METHOD Initialization : BOOL
VAR_INPUT
	_Testmode	: BOOL;
END_VAR

VAR
	bConfig: BOOL;
END_VAR
(*
_tmrT0(IN:=TRUE,PT:=T#0.2S);
LoadCell.i_bCmd_Tara:= NOT _tmrT0.Q  ;
Initialization	:= AssRoller.Initialization() AND _tmrT0.Q ;
SamplingWeight	:=0;
Cyl_NGPurge.qExtendCoil	:= FALSE;
Roller_Purge.qRun:= FALSE;
Motor_shock.qRun	:= FALSE;
Motor_shock.qSign	:= FALSE;
Cyl_ShockStop.qExtendCoil:= FALSE;
*)

_bInitialScan:=TRUE;

CASE nInitiStep OF
	0:		
		LoadCell.GetTara();
		_tmrT0(IN:=FALSE);
		strText:='ORG : Initial ';
		Cyl_NGPurge.qExtendCoil		:= FALSE;
		Roller_Purge.qRun			:= FALSE;
		Motor_shock.qRun			:= FALSE;
		Motor_shock.qSign			:= FALSE;
		Cyl_ShockStop.qExtendCoil	:= FALSE;		
		nInitiStep						:= 5;
	5:
		bConfig			:=TRUE;
		IF Sen_TFLoadIn THEN
			bConfig			:=FALSE;
			EventLogger.eEventType		:= 3;
			EventLogger.strEventText	:= 'TF Sensor Error ';	
			EventLogger();					
		END_IF		
			
		IF bConfig THEN
			nInitiStep	:= 10;
			strText:='ORG : Runing ';
			ELSE
			strText:='ORG : Failed ';
			nInitiStep	:= 50;
		END_IF	
	10:
		IF AssRoller.Initialization() THEN
			strText		:='ORG : Done ';
			nInitiStep	:= 20;
		END_IF;		
	20:
		Initialization	:= TRUE;
	
END_CASE;
END_METHOD

{warning 'add property implementation'}
PROPERTY NoEntry : BOOL
GET
END_GET
END_PROPERTY

{warning 'add method implementation '}
METHOD Pause : BOOL
END_METHOD

METHOD Process : BOOL
VAR_INPUT
	bHlatMode	: BOOL;
END_VAR

VAR
	bStoppedComv: BOOL;
END_VAR
_bProcessScan:= TRUE;
//判斷 

CASE nStep OF
	0:
		tmrLoadcell(IN:= FALSE);
		_tmrT0(IN:=FALSE);
		AssRoller.Roller();
		strText:= 'Waiting';
		IF Sen_TFLoadIn THEN
			nStep := 5;
		END_IF
	5:
		strText:= 'Loadind and Stop';
		AssRoller.Roller();
		IF NOT Sen_TFLoadIn THEN
			SamplingWeight	:= 0;
			nStep := 10;
		END_IF	
	10:		
		strText:= 'Weight Check!';
		tmrLoadcell(IN:= TRUE,PT:=T#1S);
		UpperWeight	:= RunParameter.PackagingWeight + RunParameter.PackagingWeightUpLimit ;
		LowerWeight := RunParameter.PackagingWeight - RunParameter.PackagingWeightLowLimit ;
		IF tmrLoadcell.Q THEN
			tmrLoadcell(IN:= FALSE,PT:=T#1S);
			SamplingWeight	:= 	LoadCell.o_rWeight;
			IF SamplingWeight >= LowerWeight AND
				SamplingWeight <= UpperWeight THEN
				strText:= 'Weight Pass!';
				bBoxPass:= TRUE;
				ELSE
				EventLogger.eEventType		:= 2;
				EventLogger.strEventText	:= 'Box Over Weight ';	
				EventLogger.strEventText	:=	CONCAT(EventLogger.strEventText,LEFT(REAL_TO_STRING(SamplingWeight),3));
				EventLogger();
				strText:= 'Box NG';
				bBoxPass:= FALSE;
			END_IF
			nStep := 15;
		END_IF
	
	15:
		
		IF nNGstep = 0 THEN
			nNGstep	:= 5;
			IF RunParameter.PackagingCheck THEN
				bStoppedComv	:= TRUE;
			END_IF
			AssRoller.Belt();
			IF Sen_NGLoadOut THEN
				nStep := 0;
			END_IF;
		END_IF
		
		
		
		
END_CASE;

CASE nNGstep OF
	0:
		strNGText	:= 'Wait BOX';
		tmrNG(IN:=FALSE,PT:=T#2S);
		Roller_Purge.qRun:= TRUE;
		IF Sen_NGLoadOut THEN
			strNGText	:= 'Active Loading';
			nNGstep := 20;
			CASE nStep OF
				0..10:
				strNGText	:= 'Up Loading';
				nNGstep := 50;
			END_CASE
		END_IF
	5:
		strNGText	:= 'TF Loading';
		AssRoller.Belt();
	
		IF Sen_NGLoadOut THEN
			nStep := 0;
			nNGstep	:= 6;
		END_IF
	6:
			IF bBoxPass THEN
				strNGText	:= 'TF LoadIn Stop';
				Roller_Purge.qRun:= FALSE;
				nStep := 0;
				IF nShackStep = 1 THEN
					strNGText	:= 'Go Shack';
					Roller_Purge.qRun:= TRUE;
					nNGstep	:= 10;
				END_IF;
				ELSE
				EventLogger.eEventType		:= 2;
				EventLogger.strEventText	:= 'NG Perge!';		
				EventLogger();		
				strNGText	:= 'TF NG Perge';
				nNGstep	:= 30;
				Roller_Purge.qRun:= FALSE;
			END_IF		

		
	10:
		IF Sen_ShockPos THEN
			strNGText	:= 'Shack ORG';
			nNGstep	:= 0;
		END_IF
	
	
	30://重量Error
		Cyl_NGPurge.qExtendCoil	:= TRUE;
		tmrNG(IN:=TRUE,PT:=T#2S);
		IF tmrNG.Q THEN
			tmrNG(IN:=FALSE);
			nStep := 0;
			Cyl_NGPurge.qExtendCoil	:= FALSE;
			nNGstep := 0;
		END_IF		
		
		
		
	50://手動投入	
		strNGText	:= '50 Man. ';
		IF Sen_ShockPos THEN
			nNGstep	:= 0;
		END_IF	
END_CASE;	
CASE nShackStep OF
	0:
		tmrshock(IN:=FALSE);
		nShackStep	:= 1;
	1:
		strShackText:='Wait Box';
		Cyl_ShockStop.qExtendCoil:= TRUE;
		tmrshock(IN:=Sen_ShockPos , PT:= RunParameter.shock_DelayTime);	
		Motor_shock.qRun	:= TRUE;
		Motor_shock.qSign	:= TRUE;
		IF tmrshock.q THEN
			strShackText:='Loading Box';
			tmrshock(IN:=FALSE);
			nShackStep	:= 5;
		END_IF
	5:
		strShackText:='Shack Box';
		Motor_shock.qSign	:= FALSE;
		tmrshock(IN:= TRUE, PT:= RunParameter.shock_HighTime);
		IF tmrshock.Q THEN
			tmrshock(IN:= FALSE);
			Motor_shock.qSign	:= TRUE;
			Cyl_ShockStop.qExtendCoil:= FALSE;
			nShackStep	:= 10;
		END_IF
	10:
		strShackText:='Load Out Box';
		tmrshock(IN:= NOT Sen_ShockPos , PT:= T#3S);				

		IF tmrshock.Q THEN
			Cyl_ShockStop.qExtendCoil:= TRUE;
			tmrshock(IN:= FALSE);
			nShackStep	:= 0;
		END_IF
		
		
END_CASE;
END_METHOD

PROPERTY Status : STRING(50)
GET
Status:= strText;
END_GET
END_PROPERTY

END_FUNCTION_BLOCK

// ---- 02_Unit/01_Customization/Ass_DualServo.TcPOU
FUNCTION_BLOCK Ass_DualServo IMPLEMENTS ITF_AutoStructCommand
VAR_INPUT
END_VAR
VAR_OUTPUT
END_VAR
VAR
	strText,strLeftText,strRightText	:STRING;
	tmrAuto	:TON:= (PT := TIME#1S0MS);
	bConfig	,_bError	:BOOL;
	_tmrT0		: TON;
	nInitiStep,nStopStep: INT;
	fb1_Stop,fb2_Stop,fbFly_Stop		:MC_Stop;
	fb1_Reset,fb2_Reset,fbFly_Reset		:MC_Reset;
	fbMC_MoveVelocityDaul: MC_MoveVelocity := (Velocity := 500);
	fbMC_GearIn: MC_GearIn;
	fbMC_GearOut: MC_GearOut;
	bDual1First,bDual2First,bDual1Done,bDual2Done	:BOOL;	
	MC_SetPositionLeft,MC_SetPositionRight,MC_SetPositionCon:MC_SetPosition;
	PreDual1Pos,PreDual2Pos	:  LREAL;
	L_Home,R_Home:MC_Home := (HomingMode := MC_HOMINGMODE.MC_ForceCalibration);
	MC_GroupReset: MC_GroupReset;
	LatchDual1Pos,LatchDual2Pos: LREAL;
	fbMC_MoveModule1,fbMC_MoveModule2	:MC_MoveModulo := (Velocity := 500);
	ConvQty	:INT;
	_bInitialScan	:BOOL;
	
	//Group
	fbMC_UngroupAllAxes	: MC_UngroupAllAxes;
	fbMC_GroupDisable	: MC_GroupDisable;
	fbAddAxis			: ARRAY[1..2] OF MC_AddAxisToGroup;
	fbMC_GroupEnable	: MC_GroupEnable;	
	fbMC_MoveAbsoluteCA_Left,fbMC_MoveAbsoluteCA_Right: MC_MoveAbsoluteCA := (Options := (GapControlMode := MC_GAP_CONTROL_MODE.mcGapControlModeFast));
	fbMC_GearInPosCA_Left,fbMC_GearInPosCA_Right		:MC_GearInPosCA;	
	nStep,nLeftStep,nRightStep,i	:INT;
	LeftLoadinQty,RifgtLoadinQty: UINT;
	bHMITriggerBtn: BOOL;
	fbMC_StopFly		:MC_Stop;
	MC_TouchProbeDual1,MC_TouchProbeDual2,MC_TouchProbeFly: MC_TouchProbe;
	TouchTriggerDual1,TouchTriggerDual2,TouchTriggerFly	:TRIGGER_REF;
	MC_AbortTrigger1,MC_AbortTrigger2					: MC_AbortTrigger;
	tmrT0,tmrT1	:TON := (ET := TIME#2S0MS);
	tmrFlyinDef	:TON;
	bPosfix	:BOOL;
	_bProcessScan: BOOL;
	_Dual1CalibrationPos , _Dual2CalibrationPos,_FlyInCalibrationPos	:LREAL;
	//
	fbSensorTrigger	:R_TRIG;
	dwSenesorTriggerTimes	:DWORD;
	
	wSlot: INT;
	bPause: BOOL;
	fRampTime: REAL;

END_VAR

Instance();
fbSensorTrigger(CLK:=Axis_FlyIn.DI.19);
IF fbSensorTrigger.Q THEN
	dwSenesorTriggerTimes	:= dwSenesorTriggerTimes+1;
END_IF



//Modhed
IF NOT _bProcessScan AND NOT _bInitialScan THEN
	MC_TouchProbeDual1.Execute	:= FALSE;
	MC_TouchProbeDual2.Execute	:= FALSE;
	strText:=strLeftText:=strRightText:='';
END_IF


IF NOT _bInitialScan THEN
	nInitiStep	:= 0;
END_IF

_bInitialScan:=FALSE;



IF NOT _bProcessScan THEN
	nStep	:= 0;
	nLeftStep	:=0;
	nRightStep	:=0;
END_IF


_bProcessScan:=FALSE;

METHOD _Clearfb : BOOL
VAR_INPUT
END_VAR
fbAddAxis[1](AxesGroup:=DualGroupRef, Axis := Axis_DualServo1, Execute := FALSE);
fbAddAxis[2](AxesGroup:=DualGroupRef, Axis := Axis_DualServo2, Execute := FALSE);
fbMC_MoveVelocityDaul(Axis:= Axis_DualServo1,Execute:= FALSE);
fbMC_GroupEnable(AxesGroup:= DualGroupRef, Execute:= FALSE);
fbMC_GroupDisable(AxesGroup:= DualGroupRef, Execute:= FALSE);	
fbMC_UngroupAllAxes(AxesGroup:= DualGroupRef,Execute:= FALSE);
fbMC_MoveAbsoluteCA_Left(Axis:= Axis_DualServo1,Execute:=FALSE);
fbMC_MoveAbsoluteCA_Right(Axis:= Axis_DualServo1,Execute:=FALSE);
_tmrT0(IN:=FALSE);
nInitiStep:=0;
nStep	:=0;
nLeftStep	:=0;
nRightStep	:=0;
		MC_AbortTrigger1(Axis:= Axis_DualServo1,TriggerInput:= TouchTriggerDual1,Execute:= FALSE);
		MC_AbortTrigger2(Axis:= Axis_DualServo2, TriggerInput:= TouchTriggerDual2,	Execute:= FALSE);
		MC_TouchProbeDual1(	Axis:= Axis_DualServo1,TriggerInput:=TouchTriggerDual1,Execute:= FALSE); 
		MC_TouchProbeDual2(	Axis:= Axis_DualServo2,TriggerInput:=TouchTriggerDual2,Execute:= FALSE); 
		
fbMC_MoveAbsoluteCA_Left(Axis:= Axis_DualServo1,Execute:=FALSE,Position:=RunParameter.Dual_LoadInPos,Velocity:=RunParameter.Dual_Velo,Gap:= RunParameter.Dual_Gap + (RunParameter.Dual_Length));
fbMC_MoveAbsoluteCA_Right(Axis:= Axis_DualServo2,Execute:=FALSE,Position:=RunParameter.Dual_LoadInPos,Velocity:=RunParameter.Dual_Velo,Gap:=fbMC_MoveAbsoluteCA_Left.Gap);
END_METHOD

METHOD ClearData : BOOL
VAR_INPUT
END_VAR
VAR
	clear	:ST_SlotData;
END_VAR
FOR i :=  1TO 5 DO
	slot[i]	:= clear	;
END_FOR;
ConvQty	:= 0;
END_METHOD

{warning 'add property implementation'}
PROPERTY Connect : STRING(50)
GET
END_GET
SET
END_SET
END_PROPERTY

PROPERTY Error : BOOL
GET
Error := _bError;
END_GET
END_PROPERTY

{warning 'add method implementation '}
METHOD ErrorClear : BOOL
END_METHOD

{warning 'add method implementation '}
METHOD FB_init : BOOL
VAR_INPUT
	(* if TRUE, the retain variables are initialized (warm start / cold start)*)
	bInitRetains	: BOOL;
	(* if TRUE, the instance afterwards gets moved into the copy code (online change)*)
	bInCopyCode	: BOOL;
END_VAR
END_METHOD

METHOD GroupAllAxes : BOOL
fbMC_GroupDisable(AxesGroup:= DualGroupRef, Execute:= FALSE);	
fbMC_UngroupAllAxes(AxesGroup:= DualGroupRef,Execute:= FALSE);

fbAddAxis[1].IdentInGroup := UDINT_TO_IDENTINGROUP(1); //X-Axis
fbAddAxis[2].IdentInGroup := UDINT_TO_IDENTINGROUP(2); //Y-Axis
fbAddAxis[1](AxesGroup:=DualGroupRef, Axis := Axis_DualServo1, Execute := TRUE);
fbAddAxis[2](AxesGroup:=DualGroupRef, Axis := Axis_DualServo2, Execute := TRUE);
fbMC_GroupEnable(AxesGroup:= DualGroupRef, Execute:= TRUE);
GroupAllAxes := fbAddAxis[1].Done AND fbAddAxis[2].Done AND fbMC_GroupEnable.Done;
END_METHOD

{warning 'add method implementation '}
METHOD HaltStepContiune : BOOL
END_METHOD

METHOD Initialization : BOOL
VAR_INPUT
	_Testmode	:BOOL;
END_VAR
_bInitialScan	:= TRUE;
TouchTriggerDual1.Mode		:= TOUCHPROBEMODE_SINGLE ; 	
TouchTriggerDual2.Mode		:= TOUCHPROBEMODE_SINGLE ; 	

CASE nInitiStep OF
0:	
		RB_CS_PickIO.cmd_bPartInPos	:=FALSE;
		fbMC_GearOut.Execute:=FALSE;
		fb1_Stop.Execute	:=FALSE;
		fbMC_MoveAbsoluteCA_Left.Execute	:= FALSE;
		fbMC_MoveAbsoluteCA_Right.Execute	:= FALSE;
		MC_TouchProbeFly.Execute:=FALSE;
		MC_TouchProbeDual1.Execute:=FALSE;
		MC_TouchProbeDual2.Execute:=FALSE;
		MC_AbortTrigger1(Axis:= Axis_DualServo1,TriggerInput:= TouchTriggerDual1,Execute:= TRUE);
		MC_AbortTrigger2(Axis:= Axis_DualServo2, TriggerInput:= TouchTriggerDual2,	Execute:= TRUE); 
		fbMC_MoveModule1(Axis:= Axis_DualServo1,Execute:= FALSE);
		fbMC_MoveModule2(Axis:= Axis_DualServo2,Execute:= FALSE);
		fbMC_MoveVelocityDaul(Axis:= Axis_DualServo1,Execute:= FALSE,Velocity:= 500);
		MC_SetPositionLeft(Axis:= Axis_DualServo1,Execute:= FALSE);
		MC_SetPositionRight(Axis:= Axis_DualServo2,Execute:= FALSE);
		MC_GroupReset(AxesGroup:= DualGroupRef,Execute:= FALSE);
		fbMC_GearOut(Slave:=Axis_DualServo2,Execute	:= FALSE);
		fbMC_GearIN(Master:=Axis_DualServo1, Slave:=Axis_DualServo2,Execute	:= FALSE);
		fbMC_MoveVelocityDaul(Axis:= Axis_DualServo1,Execute:= FALSE);
		fbMC_GroupDisable(AxesGroup:= DualGroupRef, Execute:= FALSE);	
		fbMC_UngroupAllAxes(AxesGroup:= DualGroupRef,Execute:= FALSE);
		fbAddAxis[1](AxesGroup:=DualGroupRef, Axis := Axis_DualServo1, Execute := FALSE);
		fbAddAxis[2](AxesGroup:=DualGroupRef, Axis := Axis_DualServo2, Execute := FALSE);
		fbMC_GroupEnable.Execute:= FALSE;	
		fbMC_GroupDisable.Execute:= FALSE;
		fbMC_UngroupAllAxes.Execute:= FALSE;

		_tmrT0(IN:=TRUE,PT:=T#0.1S);
		nStopStep			:= 0;
		strText:='ORG : Initial ';
		IF _tmrT0.Q THEN
			ClearData();
			_tmrT0(IN:=FALSE);
			nInitiStep	:= 1;
		END_IF;
1:

	_tmrT0(IN:= NOT _tmrT0.Q ,PT:= T#1S);
	CASE Axis_DualServo1.Status.MotionState OF
		MC_AXISSTATE_UNDEFINED:
			;
		MC_AXISSTATE_DISABLED:
			Axis_DualServo1.ServoOn();
		MC_AXISSTATE_STANDSTILL:
			;
		MC_AXISSTATE_ERRORSTOP:
			Axis_DualServo1.Reset();
		MC_AXISSTATE_DISCRETEMOTION:
			Axis_DualServo1.Reset();
		MC_AXISSTATE_CONTINOUSMOTION:
			Axis_DualServo1.Stop();
		MC_AXISSTATE_SYNCHRONIZEDMOTION	:
		;
	END_CASE

	CASE Axis_DualServo2.Status.MotionState OF
		MC_AXISSTATE_UNDEFINED:
			;
		MC_AXISSTATE_DISABLED:
			Axis_DualServo2.ServoOn();
		MC_AXISSTATE_STANDSTILL:
			;
		MC_AXISSTATE_ERRORSTOP:
			Axis_DualServo2.Reset();
		MC_AXISSTATE_DISCRETEMOTION:
			Axis_DualServo2.Reset();
		MC_AXISSTATE_CONTINOUSMOTION:
			Axis_DualServo2.Stop();
		MC_AXISSTATE_SYNCHRONIZEDMOTION	:
			fbMC_GearOut( Slave:=Axis_DualServo2,Execute:= TRUE);
	END_CASE	
	CASE Axis_FlyIn.Status.MotionState OF
		MC_AXISSTATE_UNDEFINED:
			;
		MC_AXISSTATE_DISABLED:
			Axis_FlyIn.ServoOn();
		MC_AXISSTATE_STANDSTILL:
			;
		MC_AXISSTATE_ERRORSTOP:
			Axis_FlyIn.Reset();

		MC_AXISSTATE_CONTINOUSMOTION:
			Axis_FlyIn.Stop();

	END_CASE
	
	
	
	IF Axis_DualServo1.Status.MotionState =MC_AXISSTATE_STANDSTILL AND Axis_DualServo2.Status.MotionState =MC_AXISSTATE_STANDSTILL AND Axis_FlyIn.Status.MotionState =MC_AXISSTATE_STANDSTILL THEN
		_tmrT0(IN:=FALSE);
		nInitiStep	:= 5;
	END_IF
	IF _tmrT0.Q THEN
		_tmrT0(IN:=FALSE);
		nInitiStep	:= 5;		
	END_IF
	
	
5:	
	bConfig			:=TRUE;
	IF NOT Axis_DualServo2.Status.StandStill THEN
		bConfig			:=FALSE;
		EventLogger.eEventType		:= 3;
		EventLogger.strEventText	:= 'Dual:ServoError ';	
		EventLogger();					
	END_IF
	IF NOT Axis_DualServo1.Status.StandStill THEN
		bConfig			:=FALSE;
		EventLogger.eEventType		:= 3;
		EventLogger.strEventText	:= 'Dual:ServoError ';		
		EventLogger();					
	END_IF
	IF NOT Axis_FlyIn.Status.StandStill THEN
		//bConfig			:=FALSE;
		EventLogger.eEventType		:= 3;
		EventLogger.strEventText	:= 'Dual:ServoError ';			
		EventLogger();					
	END_IF
	
	IF bConfig THEN
		_tmrT0(IN:= FALSE);
		nInitiStep:= nInitiStep + 5 ;
		strText:='ORG:Syc. ';
		ELSE
		OP.bInitialSign		:=FALSE;
		OP.xInitialRuning	:=FALSE;
		nInitiStep := nInitiStep +100;	
		strText:='ORG:Error Stop ';
	END_IF	
	
10://軸同步 
	bDual1First:=bDual2First:=bDual1Done:=bDual2Done	:=FALSE;
	fbMC_GearIn(Master:= Axis_DualServo1, Slave:=Axis_DualServo2 ,Execute	:= TRUE );
	IF fbMC_GearIn.InGear THEN
		fbMC_GearIn.Execute:=FALSE;	
		nInitiStep	:= 11;
	END_IF	
	IF fbMC_GearIn.Error THEN
		fbMC_GearIn.Execute:=FALSE;	
		nInitiStep	:= 99;
	END_IF	
11:
	fbMC_GearOut.Execute:=FALSE;
	MC_TouchProbeDual1.Execute:= TRUE;	
	MC_TouchProbeDual2.Execute:= TRUE;	
	IF MC_TouchProbeDual1.Busy AND MC_TouchProbeDual2.Busy THEN
		nInitiStep	:= 15;
	END_IF	
	
15://馬達啟動 
	strText:='ORG:Act.';
	fbMC_MoveVelocityDaul(Axis:= Axis_DualServo1,Execute:= TRUE,Velocity:= 500);
	IF fbMC_MoveVelocityDaul.Busy THEN
		nInitiStep	:= 20;
	END_IF

20:	//感測sensor
		MC_TouchProbeDual1(
	Axis:= Axis_DualServo1, 
	TriggerInput:=TouchTriggerDual1 , 
	Execute:= TRUE, 
	WindowOnly:= , 
	FirstPosition:= , 
	LastPosition:= , 
	Done=> , 
	Busy=> , 
	CommandAborted=> , 
	Error=> , 
	ErrorID=> , 
	RecordedPosition=> , 
	RecordedData=> );
		MC_TouchProbeDual2(
	Axis:= Axis_DualServo2, 
	TriggerInput:=TouchTriggerDual2 , 
	Execute:= TRUE, 
	WindowOnly:= , 
	FirstPosition:= , 
	LastPosition:= , 
	Done=> , 
	Busy=> , 
	CommandAborted=> , 
	Error=> , 
	ErrorID=> , 
	RecordedPosition=> , 
	RecordedData=> );	
	IF MC_TouchProbeDual1.Done AND NOT bDual1Done THEN
		LatchDual1Pos	:=  MC_TouchProbeDual1.RecordedData.RecordedPosition;
		bDual1Done	:= TRUE;
		IF NOT bDual2First THEN
			bDual1First	:= TRUE;
		END_IF
	END_IF

	IF MC_TouchProbeDual2.Done AND NOT bDual2Done THEN
		LatchDual2Pos	:=  MC_TouchProbeDual2.RecordedData.RecordedPosition;
		bDual2Done	:= TRUE;
		IF NOT bDual1First THEN
			bDual2First	:= TRUE;
		END_IF
	END_IF
		
	IF bDual1Done AND bDual2Done THEN
		MC_TouchProbeDual1.Execute:=FALSE;
		MC_TouchProbeDual2.Execute:=FALSE;
		nInitiStep:=25;
	END_IF	
25:
	strText:='ORG : GetPosition ';
	IF Axis_DualServo1.Status.MotionState = MC_AXISSTATE_STANDSTILL THEN
		fbMC_GearOut.Execute:=TRUE;
		IF NOT Axis_DualServo2.Status.Coupled THEN
			fbMC_GearOut.Execute:=FALSE;
			nInitiStep		:= nInitiStep+5;
		END_IF;
			
		ELSIF Axis_DualServo1.Status.MotionState = MC_AXISSTATE_STOPPING THEN
			fb1_Stop.Execute:=FALSE;
		ELSE
			fb1_Stop.Execute:=TRUE;
	END_IF		
30:

	fbMC_MoveVelocityDaul(Axis:= Axis_DualServo1,Execute:= FALSE);
	MC_SetPositionLeft.Position	:= Axis_DualServo1.NcToPlc.ActPos - LatchDual1Pos- Setting_Dual1_ORG_Offset
 ;
	MC_SetPositionRight.Position:= Axis_DualServo2.NcToPlc.ActPos - LatchDual2Pos- Setting_Dual2_ORG_Offset;
	MC_SetPositionLeft(Axis:= Axis_DualServo1,Execute:= TRUE);
	MC_SetPositionRight(Axis:= Axis_DualServo2,Execute:= TRUE);
	MC_SetPositionCon(Axis:= Axis_FlyIn,Execute:= TRUE);
	IF MC_SetPositionLeft.Done AND MC_SetPositionRight.Done AND MC_SetPositionCon.Done THEN
		nInitiStep		:= nInitiStep+1;
	END_IF

31:
	L_Home(Axis:= Axis_DualServo1,Execute:= TRUE);
	R_Home(Axis:= Axis_DualServo2,Execute:= TRUE);
	IF L_Home.Done AND L_Home.Done THEN
		nInitiStep		:= 35;
		IF _Testmode THEN
			nInitiStep		:= 50;
		END_IF
	END_IF
35:
	MC_GroupReset(
	AxesGroup:= DualGroupRef, 
	Execute:= TRUE, 
	Done=> , 
	Busy=> , 
	Error=> , 
	ErrorId=> );
	IF MC_GroupReset.Done THEN
		nInitiStep		:= nInitiStep +1 ;	
	END_IF;

 
36:
	IF GroupAllAxes() THEN
		nInitiStep		:= 40;
	END_IF
40:
	(*
	EventLogger.eEventType		:= 1;
	EventLogger.strEventText	:= 'DualServo ORG Done';	
	EventLogger();
	*)
	nInitiStep		:= nInitiStep+5;	
45:
	strText:='ORG : Done ';
	Initialization:= TRUE;
	
50://test mode
	fbMC_MoveModule1(Axis:= Axis_DualServo1,Execute:= TRUE);
	fbMC_MoveModule2(Axis:= Axis_DualServo2,Execute:= TRUE,Position:= fbMC_MoveModule1.Position);
	IF fbMC_MoveModule1.Done AND fbMC_MoveModule2.Done THEN
		nInitiStep		:= 45;	
	END_IF
	
99..199:
;
END_CASE;
END_METHOD

ACTION Instance:
TouchTriggerFly.EncoderID  := Axis_FlyIn.DriveAddress.NcEncoderId ;
TouchTriggerFly.TouchProbe := TouchProbe1 ; 
TouchTriggerFly.SignalSource:= SignalSource_Input1;
TouchTriggerFly.Edge:=RisingEdge;
TouchTriggerFly.Mode:= TOUCHPROBEMODE_CONTINOUS  ; 
TouchTriggerDual1.EncoderID  := Axis_DualServo1.DriveAddress.NcEncoderId ;
TouchTriggerDual1.TouchProbe := TouchProbe1 ; 
TouchTriggerDual1.SignalSource:= SignalSource_Input1;
TouchTriggerDual1.Edge:=RisingEdge;
TouchTriggerDual2.EncoderID  := Axis_DualServo2.DriveAddress.NcEncoderId ;
TouchTriggerDual2.TouchProbe := TouchProbe1 ; 
TouchTriggerDual2.SignalSource:= SignalSource_Input1;
TouchTriggerDual2.Edge		:=RisingEdge;
fb1_Stop(Axis	:=Axis_DualServo1);
fbMC_GearOut(Slave:=Axis_DualServo2);

MC_TouchProbeFly(Axis:= Axis_FlyIn, TriggerInput:=TouchTriggerFly);
MC_TouchProbeDual1(	Axis:= Axis_DualServo1,TriggerInput:=TouchTriggerDual1); 
MC_TouchProbeDual2(	Axis:= Axis_DualServo2,TriggerInput:=TouchTriggerDual2);
fbMC_MoveAbsoluteCA_Left(Axis:= Axis_DualServo1,Gap:= RunParameter.Dual_Gap+RunParameter.Dual_Length ,Direction:=mcDirectionPositive);
fbMC_MoveAbsoluteCA_Right(Axis:= Axis_DualServo2,Gap:= RunParameter.Dual_Gap+RunParameter.Dual_Length,Direction:=mcDirectionPositive);
fbMC_GroupEnable(AxesGroup:= DualGroupRef);	
fbMC_GroupDisable(AxesGroup:= DualGroupRef);
fbMC_UngroupAllAxes(AxesGroup:= DualGroupRef);	

//
IF MC_TouchProbeDual1.Error  THEN
	MC_TouchProbeDual1.Execute :=FALSE;
END_IF
IF MC_TouchProbeDual2.Error  THEN
	MC_TouchProbeDual2.Execute :=FALSE;
END_IF
END_ACTION

PROPERTY NoEntry : BOOL
GET
END_GET
END_PROPERTY

{warning 'add method implementation '}
METHOD Pause : BOOL
END_METHOD

METHOD Process : BOOL
VAR_INPUT
	bHlatMode	: BOOL;
END_VAR
_bProcessScan	:= TRUE;
TouchTriggerDual1.Mode		:= TOUCHPROBEMODE_CONTINOUS ; 	
TouchTriggerDual2.Mode		:= TOUCHPROBEMODE_CONTINOUS ; 	
fRampTime					:= RunParameter.Fly_Disdance	/RunParameter.Fly_Velo;



CASE  nStep OF
	0:
		wSlot	:=0;
		
		MC_SetPositionCon(Axis:=Axis_FlyIn,Execute:=FALSE);
		fbMC_StopFly(Axis:= Axis_FlyIn,Execute:= FALSE);
		IF DualGroupRef.NcToPlc.Common.GroupStatus.State = mcGroupStateStandby AND DualGroupRef.NcToPlc.Common.GroupAxesCount = 2 THEN
			OP.bCycleStep	:= FALSE;
			ClearData();
			nStep	:= 1;			
		END_IF	
	1:
		MC_SetPositionCon(Axis:=Axis_FlyIn,Execute:=TRUE,Position:= 0);
		IF 	MC_SetPositionCon.Done THEN
			MC_TouchProbeFly.Execute	:= TRUE;
			nStep	:= 2;	
		END_IF
	2:
		tmrFlyinDef(IN:=FALSE);
		IF MC_TouchProbeFly.Busy THEN
			_FlyInCalibrationPos	:= MC_TouchProbeFly.RecordedData.RecordedPosition;
			nStep	:=5;	
		END_IF;	
	5:
		strText	:= 'AutoFeed';
		IF NOT bPause THEN
			strText	:= 'Pause';
			Axis_FlyIn.MoveVelocity(RunParameter.Fly_Velo,1);
		END_IF;
		//feedin def
		tmrFlyinDef(PT:=T#0.2S);
		IF tmrFlyinDef.IN THEN
			_FlyInCalibrationPos	:= MC_TouchProbeFly.RecordedData.RecordedPosition;
		END_IF
		IF tmrFlyinDef.Q THEN
			tmrFlyinDef.IN	:= FALSE;
		END_IF
		IF _FlyInCalibrationPos <>  MC_TouchProbeFly.RecordedData.RecordedPosition THEN
			tmrFlyinDef.IN	:= TRUE;
			_FlyInCalibrationPos	:= MC_TouchProbeFly.RecordedData.RecordedPosition;
			ResInData(_FlyInCalibrationPos);
		END_IF
	

		//auto test tool
		IF Hmi_bDualFeedTest THEN
			ResInData(Axis_FlyIn.NcToPlc.ActPos);
			Hmi_bDualFeedTest	:=FALSE;
		END_IF
		
		tmrAuto(IN:=Hmi_bDualAutoTest AND NOT tmrAuto.Q AND Motor_LoadIn.qRun,PT:=Hmi_bDualAutoTestTime );
		
		IF  tmrAuto.q AND ConvQty < 1 THEN
			ResInData(Axis_FlyIn.NcToPlc.ActPos);		
		END_IF
		//////////////////////
		
		IF OP.bStop_Sign THEN
			fbMC_StopFly.Execute:= TRUE;
			nStep:= 10;
		END_IF
		
		IF slot[1].ScanIn AND NOT slot[1].LoadIn THEN
			IF  Axis_FlyIn.NcToPlc.ActPos>slot[1].GearInPosition THEN
				slot[1].LoadIn	:=TRUE;
			END_IF
		END_IF

		
	10:
		;
END_CASE
	
tmrT0();
CASE nLeftStep OF
	0:
		strLeftText:='Para Set';
		MC_TouchProbeDual1.Execute:= TRUE;
		IF MC_TouchProbeDual1.Busy THEN
			_Dual1CalibrationPos	:= MC_TouchProbeDual1.RecordedData.RecordedPosition;
			nLeftStep	:=1;	
		END_IF;			
	
	
	1:	
			strLeftText:='P1 moving';
			fbMC_MoveAbsoluteCA_Left.Execute	:=TRUE;
			fbMC_MoveAbsoluteCA_Left.Position	:= RunParameter.Dual_LoadInPos;
			fbMC_MoveAbsoluteCA_Left.Velocity	:=RunParameter.Dual_Velo;
			fbMC_MoveAbsoluteCA_Left.Acceleration	:= 15000;
			fbMC_MoveAbsoluteCA_Left.Deceleration	:= 15000;
			fbMC_MoveAbsoluteCA_Left.Jerk			:= 50000;
			LeftLoadinQty	:=0;
			nLeftStep		:= 5;

	5:
		IF Axis_DualServo1.Status.NotMoving THEN
			strLeftText:='P1 Coupled';
			ELSE
			strLeftText:='P1 moving';
		END_IF;	
	
		IF fbMC_MoveAbsoluteCA_Left.Done THEN
			strLeftText:='P1 Pos';
			fbMC_MoveAbsoluteCA_Left.Execute	:= FALSE;
			nLeftStep	:=10;
		END_IF
	10: 
		strLeftText:='P1 Pos';
		strLeftText	:= CONCAT(strLeftText,UINT_TO_STRING(LeftLoadinQty));	
		IF slot[1].LoadIn THEN
			LeftLoadinQty	:= 	LeftLoadinQty+1;
			ResOut();
			IF LeftLoadinQty < RunParameter.Dual_LoadInQty[wSlot] THEN
				strLeftText:='P1 Next Pos';
				strLeftText	:= CONCAT(strLeftText,UINT_TO_STRING(LeftLoadinQty));
				fbMC_MoveAbsoluteCA_Left.Execute	:= TRUE;
				fbMC_MoveAbsoluteCA_Left.Position	:= fbMC_MoveAbsoluteCA_Left.Position + RunParameter.Dual_ModulePitchLength;
				fbMC_MoveAbsoluteCA_Left.Velocity	:= 1500;
				//fbMC_MoveAbsoluteCA_Left.Velocity	:= RunParameter.Dual_ModulePitchLength / (fRampTime*0.5);		
				nLeftStep	:= 5;
				ELSE
				wSlot								:= wSlot + 1;
				IF RunParameter.Dual_LoadInQty[wSlot] = 0 THEN
					wSlot	:= 0;
				END_IF
				fbMC_MoveAbsoluteCA_Left.Execute		:= TRUE;
				fbMC_MoveAbsoluteCA_Left.Position		:= RunParameter.Dual_LoadOutPos;	
				fbMC_MoveAbsoluteCA_Left.Velocity		:= RunParameter.Dual_Velo;
				fbMC_MoveAbsoluteCA_Left.Acceleration	:= Parameter_PERSISTENT.Setting_DualServoAcc;
				fbMC_MoveAbsoluteCA_Left.Deceleration	:= Parameter_PERSISTENT.Setting_DualServoDec;
				fbMC_MoveAbsoluteCA_Left.Jerk			:= Parameter_PERSISTENT.Setting_DualServoJerk;			
				strLeftText:='P2 moving';			
				nLeftStep	:= 20;					
			END_IF;
		END_IF	



	20://裝完 
		IF Axis_DualServo1.Status.NotMoving THEN
			strLeftText:='P2 Coupled';
			ELSE
			strLeftText:='P2 moving';	
		END_IF
	
		IF fbMC_MoveAbsoluteCA_Left.Done THEN
			strLeftText:='P2 Pos Call RB';	
			fbMC_MoveAbsoluteCA_Left.Execute	:= FALSE;
			nLeftStep	:= 24;
			RB_CS_PickIO.cmd_bPartInPos	:= TRUE;

		END_IF		
	24://RB輸出通知 
		IF RB_CS_PickIO.fb_bPackFinish	THEN
			RB_CS_PickIO.cmd_bPartInPos	:= FALSE;
			nLeftStep	:= 25;
		END_IF		
			IF Hmi_bPickFeedTest THEN
				RB_CS_PickIO.cmd_bPartInPos	:= FALSE;
				Hmi_bPickFeedTest			:=FALSE;
				nLeftStep					:= 29;	
			END_IF
	25:
		IF NOT RB_CS_PickIO.fb_bPackFinish	THEN
			nLeftStep	:= 29;
		END_IF	

	
	29://RB輸出通知

			IF NOT RunParameter.Dual_TwiceClip THEN
				nLeftStep		:= 1;
				ELSE
				strLeftText:='P3 moving';
				nLeftStep		:= 30;
				fbMC_MoveAbsoluteCA_Left.Execute	:=TRUE;
				fbMC_MoveAbsoluteCA_Left.Position	:= RunParameter.Dual_LoadOutSecPos;
			END_IF;	

	30:
	
		IF fbMC_MoveAbsoluteCA_Left.Done THEN
			strRightText:='P3 Pos Call RB';
			fbMC_MoveAbsoluteCA_Left.Execute	:= FALSE;
			RB_CS_PickIO.cmd_bPartInPos	:= TRUE;
			nLeftStep	:=31;
		END_IF			
		
	31:
		IF Hmi_bPickFeedTest THEN
			RB_CS_PickIO.cmd_bPartInPos	:= FALSE;
			Hmi_bPickFeedTest			:=FALSE;
			nLeftStep					:= 1;	
		END_IF	
		IF RB_CS_PickIO.fb_bPackFinish	THEN
			RB_CS_PickIO.cmd_bPartInPos	:= FALSE;
			nLeftStep	:= 32;
		END_IF			
	32:	
		IF NOT RB_CS_PickIO.fb_bPackFinish	THEN
			nLeftStep	:= 1;
		END_IF		
	
END_CASE

CASE nRightStep OF
	0:
		strRightText:='Para Set';
		MC_TouchProbeDual2.Execute:= TRUE;
		IF MC_TouchProbeDual2.Busy THEN
			_Dual2CalibrationPos	:= MC_TouchProbeDual2.RecordedData.RecordedPosition;
			nRightStep	:=1;	
		END_IF;			
	1:
			strRightText:='P1 moving';
			fbMC_MoveAbsoluteCA_Right.Execute:= TRUE;
			fbMC_MoveAbsoluteCA_Right.Position	:= RunParameter.Dual_LoadInPos;
			fbMC_MoveAbsoluteCA_Right.Velocity	:=RunParameter.Dual_Velo;
			fbMC_MoveAbsoluteCA_Right.Acceleration	:= 15000;
			fbMC_MoveAbsoluteCA_Right.Deceleration	:= 15000;
			fbMC_MoveAbsoluteCA_Right.Jerk			:= 50000;
			RifgtLoadinQty	:=0;
			nRightStep		:= 5;

	5:
		IF Axis_DualServo2.Status.NotMoving THEN
			strRightText:='P1 Coupled';
			ELSE
			strRightText:='P1 moving';
		END_IF;			
		IF fbMC_MoveAbsoluteCA_Right.Done THEN
			strRightText:='P1 Pos';
			fbMC_MoveAbsoluteCA_Right.Execute	:= FALSE;
			nRightStep	:=10;
		END_IF
	10: 
				strRightText	:='P1 Pos';
				strRightText	:= CONCAT(strRightText,UINT_TO_STRING(RifgtLoadinQty));	
		IF slot[1].LoadIn THEN
			RifgtLoadinQty	:= 	RifgtLoadinQty+1;
			ResOut();
			IF RifgtLoadinQty < RunParameter.Dual_LoadInQty[wSlot] THEN
				fbMC_MoveAbsoluteCA_Right.Execute	:= TRUE;
				fbMC_MoveAbsoluteCA_Right.Position	:= fbMC_MoveAbsoluteCA_Right.Position + RunParameter.Dual_ModulePitchLength;				
				fbMC_MoveAbsoluteCA_Right.Velocity	:= 1500;		
				nRightStep	:= 5;
				ELSE
				wSlot								:= wSlot + 1;
				IF RunParameter.Dual_LoadInQty[wSlot] = 0 THEN
					wSlot	:= 0;
				END_IF
				fbMC_MoveAbsoluteCA_Right.Execute	:= TRUE;
				fbMC_MoveAbsoluteCA_Right.Position	:= RunParameter.Dual_LoadOutPos;	
				fbMC_MoveAbsoluteCA_Right.Velocity		:=RunParameter.Dual_Velo;
				fbMC_MoveAbsoluteCA_Right.Acceleration	:= Parameter_PERSISTENT.Setting_DualServoAcc;
				fbMC_MoveAbsoluteCA_Right.Deceleration	:= Parameter_PERSISTENT.Setting_DualServoDec;
				fbMC_MoveAbsoluteCA_Right.Jerk			:= Parameter_PERSISTENT.Setting_DualServoJerk;
				strRightText:='P2 moving';
				nRightStep	:= 20;					
			END_IF;

		END_IF	

	20://裝完
		IF Axis_DualServo2.Status.NotMoving THEN
			strRightText:='P2 Coupled';
			ELSE
			strRightText:='P2 moving';	
		END_IF
	
	
		IF fbMC_MoveAbsoluteCA_Right.Done THEN
			strRightText:='P2 Pos Call RB';	
			fbMC_MoveAbsoluteCA_Right.Execute	:= FALSE;
			RB_CS_PickIO.cmd_bPartInPos	:= TRUE;
			nRightStep	:= 24;
		END_IF		
	24://RB輸出通知 
		IF RB_CS_PickIO.fb_bPackFinish	THEN
			RB_CS_PickIO.cmd_bPartInPos	:= FALSE;
			nRightStep	:= 25;
		END_IF		
			IF Hmi_bPickFeedTest THEN
				RB_CS_PickIO.cmd_bPartInPos	:= FALSE;
				Hmi_bPickFeedTest			:=FALSE;
				nRightStep					:= 29;	
			END_IF
	25:
		IF NOT RB_CS_PickIO.fb_bPackFinish	THEN
			nRightStep	:= 29;
		END_IF		
	
				
	29:
			IF NOT RunParameter.Dual_TwiceClip THEN
				nRightStep		:= 1;
				ELSE
				strRightText:='P3 moving';
				nRightStep		:= 30;
				fbMC_MoveAbsoluteCA_Right.Execute	:=TRUE;
				fbMC_MoveAbsoluteCA_Right.Position	:= RunParameter.Dual_LoadOutSecPos;
			
			END_IF;	
	30:
	
		IF fbMC_MoveAbsoluteCA_Right.Done THEN
			strRightText:='P3 Pos Call RB';
			fbMC_MoveAbsoluteCA_Right.Execute	:= FALSE;
			RB_CS_PickIO.cmd_bPartInPos	:= TRUE;
			nRightStep	:=31;
		END_IF			
	31:
		IF Hmi_bPickFeedTest THEN
			RB_CS_PickIO.cmd_bPartInPos	:= FALSE;
			Hmi_bPickFeedTest			:=FALSE;
			nRightStep					:= 1;	
		END_IF	
		IF RB_CS_PickIO.fb_bPackFinish	THEN
			RB_CS_PickIO.cmd_bPartInPos	:= FALSE;
			nRightStep	:= 32;
		END_IF			
	32:	
		IF NOT RB_CS_PickIO.fb_bPackFinish	THEN
			nRightStep	:= 1;
		END_IF		

END_CASE

CASE nStopStep OF
	0:
		Motor_LoadIn.qRun	:= TRUE;
		Cyl_FlyIn_Pass		:= TRUE;
		(*
		IF nLeftStep < 20 THEN
			IF fbMC_MoveAbsoluteCA_Left.Busy AND Axis_DualServo1.Status.NotMoving THEN
				Motor_LoadIn.qRun	:= FALSE;
				Cyl_FlyIn_Pass		:= FALSE;
			END_IF; 
			IF nRightStep < 5 THEN
				Motor_LoadIn.qRun	:= FALSE;
				Cyl_FlyIn_Pass		:= FALSE;
			END_IF
			IF nRightStep = 10 THEN
				Motor_LoadIn.qRun	:= TRUE;
				Cyl_FlyIn_Pass		:= TRUE;
			END_IF				
			
		END_IF;
		
		IF nRightStep < 20 THEN
			IF fbMC_MoveAbsoluteCA_Right.Busy AND Axis_DualServo2.Status.NotMoving THEN
				Motor_LoadIn.qRun	:= FALSE;
				Cyl_FlyIn_Pass		:= FALSE;
			END_IF; 
			IF nLeftStep < 5 THEN
				Motor_LoadIn.qRun	:= FALSE;
				Cyl_FlyIn_Pass		:= FALSE;
			END_IF
			IF nLeftStep = 10 THEN
				Motor_LoadIn.qRun	:= TRUE;
				Cyl_FlyIn_Pass		:= TRUE;
			END_IF			
		END_IF
	//IF nLeftStep < 20 AND nRightStep < 20 THEN
	//	Motor_LoadIn.qRun	:= TRUE;
	//	Cyl_FlyIn_Pass		:= TRUE;
	//END_IF
*)
END_CASE
//_label1 : ;
END_METHOD

METHOD ResInData :BOOL;
VAR_INPUT
	Pos	: LREAL;
END_VAR

IF ConvQty < 5 THEN
ConvQty:= ConvQty+1;
slot[ConvQty].ScanIn			:= TRUE;
slot[ConvQty].LatchPosition		:= Pos;
slot[ConvQty].GearInPosition	:= Pos + RunParameter.Fly_Disdance;
END_IF;
END_METHOD

METHOD ResOut
VAR_IN_OUT
END_VAR
IF ConvQty <>0 THEN
	FOR i := 1 TO ConvQty BY 1 DO
		slot[i]:= slot[i+1];
	END_FOR
	ConvQty	:= ConvQty - 1;
END_IF;
END_METHOD

METHOD RingTest : BOOL
VAR_INPUT
END_VAR
END_METHOD

PROPERTY Status : STRING(50)
GET
END_GET
END_PROPERTY

METHOD STOP : BOOL
VAR_INPUT
END_VAR
IF Axis_FlyIn.Status.Moving THEN
	Axis_FlyIn.Stop();	
END_IF

IF Axis_DualServo1.Status.Moving THEN
	Axis_DualServo1.Stop();	
END_IF
END_METHOD

METHOD UngroupAllAxes : BOOL
fbMC_GroupDisable.Execute:= TRUE;
IF fbMC_GroupDisable.Done THEN
	fbMC_UngroupAllAxes.Execute:= TRUE;
END_IF;
fbMC_GroupEnable.Execute:= FALSE;
fbAddAxis[1](AxesGroup:=DualGroupRef, Axis := Axis_DualServo1, Execute := FALSE);
fbAddAxis[2](AxesGroup:=DualGroupRef, Axis := Axis_DualServo2, Execute := FALSE);

	
	
UngroupAllAxes :=fbMC_UngroupAllAxes.Done AND fbMC_GroupDisable.Done AND DualGroupRef.NcToPlc.CA.Common.GroupAxesCount = 0;
END_METHOD

END_FUNCTION_BLOCK

// ---- 02_Unit/01_Customization/Ass_Openbox.TcPOU
FUNCTION_BLOCK Ass_Openbox IMPLEMENTS ITF_AutoStructCommand
VAR_INPUT
END_VAR
VAR_OUTPUT
END_VAR
VAR
	strText	:STRING;
	i	:INT;
	MC_MoveAbsolute		: MC_MoveAbsolute;
	MC_Home				: MC_Home;
	_bProcessScan,_bInitialScan: BOOL;
	_bHalt , _bError,_bHaltPause: BOOL;
	nStep,nStt,nInitiStep	: INT;
	nNextStep		: INT;
	tmrClear		:TON;
	temp: DWORD;
	tmrloadIn,tmrloadIn2,tmrDelay: TON;
	wPunchcounter	:INT;
	_tmrT0: TON;
END_VAR

MC_Home(Axis:= Axis_BoxPullOut,bCalibrationCam := NOT Sen_AxisBoxORG);

IF NOT _bInitialScan THEN
	nInitiStep	:= 0;
END_IF

_bInitialScan:=FALSE;



IF NOT _bProcessScan THEN
	nNextStep	:= 0;
	nStep		:= 0;
END_IF

_bProcessScan	:=FALSE;

{warning 'add property implementation'}
PROPERTY Connect : STRING(50)
GET
END_GET
SET
END_SET
END_PROPERTY

METHOD INTERNAL Cyl_Safe : BOOL
VAR_INPUT
END_VAR
Cyl_Safe	:= Cyl_AxisBoxCatch.iOriginSensor AND Cyl_Axis90.iOriginSensor AND
				Cyl_AxisBottom.iOriginSensor AND Cyl_BoxSideBottom.iOriginSensor AND 	
				Cyl_BoxSidePitch.iOriginSensor	AND Cyl_BeltBottom.iOriginSensor ;
END_METHOD

{warning 'add property implementation'}
PROPERTY Error : BOOL
GET
END_GET
END_PROPERTY

{warning 'add method implementation '}
METHOD ErrorClear : BOOL
END_METHOD

{warning 'add method implementation '}
METHOD FB_init : BOOL
VAR_INPUT
	(* if TRUE, the retain variables are initialized (warm start / cold start)*)
	bInitRetains	: BOOL;
	(* if TRUE, the instance afterwards gets moved into the copy code (online change)*)
	bInCopyCode	: BOOL;
END_VAR
END_METHOD

METHOD HaltStepContiune : BOOL
nStep:= nNextStep;
END_METHOD

METHOD Initialization : BOOL
VAR_INPUT
	_Testmode	:BOOL;	//OOP Var
END_VAR
VAR
	bConfig: BOOL;
END_VAR
_bInitialScan	:= TRUE;
//初始化部屬 
//	IF Axis_BoxPullOut.Status.Error AND nInitiStep <> 100 THEN
//		nInitiStep:= 99;
//	END_IF
	
CASE nInitiStep OF
	0:
		_tmrT0(IN:=FALSE);
		strText:='ORG : Initial ';
		MC_Home.Execute:=FALSE;
		MC_MoveAbsolute(Axis:= Axis_BoxPullOut,Execute:=FALSE);
			
		Vacm_AxisCatchBox				:=FALSE;
		Cyl_AxisBoxCatch.qExtendCoil	:=FALSE;
		Cyl_Axis90.qExtendCoil			:=FALSE;
		Cyl_AxisBottom.qExtendCoil		:=FALSE;

		Vacm_Axis90						:=FALSE;
		Cyl_BoxSideBottom.qExtendCoil	:=FALSE;
		Cyl_BoxSidePitch.qExtendCoil	:=FALSE;
		
		Cyl_BeltBottom.qExtendCoil		:=FALSE;
		
		IF Cyl_Safe() THEN
			nInitiStep	:= 1;
		END_IF
	1:

	_tmrT0(IN:= NOT _tmrT0.Q ,PT:= T#1S);
	CASE Axis_BoxPullOut.Status.MotionState OF
		MC_AXISSTATE_UNDEFINED:
			;
		MC_AXISSTATE_DISABLED:
			IF Axis_BoxPullOut.Status.Error THEN
				Axis_BoxPullOut.Reset();
				ELSE
				Axis_BoxPullOut.ServoOn();
			END_IF;
		MC_AXISSTATE_STANDSTILL:
			;
		MC_AXISSTATE_ERRORSTOP:
			Axis_BoxPullOut.Reset();
		MC_AXISSTATE_CONTINOUSMOTION:
			Axis_BoxPullOut.Stop();
		MC_AXISSTATE_SYNCHRONIZEDMOTION	:
		;
	END_CASE
	
	IF Axis_BoxPullOut.Status.MotionState =MC_AXISSTATE_STANDSTILL THEN
		_tmrT0(IN:=FALSE);
		nInitiStep	:= 5;
	END_IF
	IF _tmrT0.Q THEN
		_tmrT0(IN:=FALSE);
		nInitiStep	:= 5;		
	END_IF

	5:
		bConfig			:=TRUE;
		IF NOT Axis_BoxPullOut.Status.StandStill THEN
			bConfig			:=FALSE;
			EventLogger.eEventType		:= 4;
			EventLogger.strEventText	:= 'BoxPullOutAxis Error ';	
			EventLogger();					
		END_IF
		
		IF bConfig THEN
			EventLogger.eEventType		:= 2;
			EventLogger.strEventText	:= 'BoxPull ORG Runing ';	
			EventLogger();
			_tmrT0(IN:= FALSE);
			nInitiStep:= nInitiStep + 5 ;
			strText:='ORG : Runing ';
			ELSE
			EventLogger.eEventType		:= 4;
			EventLogger.strEventText	:= 'Exceptions Cause interruptions!! ';	
			EventLogger();
			OP.bInitialSign		:=FALSE;
			OP.xInitialRuning	:=FALSE;
			nInitiStep := nInitiStep +100;	
			strText:='ORG : Failed ';
		END_IF	
		
	10:
		IF NOT Axis_BoxPullOut.Status.Homed THEN
			strText:='ORG : Runing ';
			nInitiStep	:= 16;
			ELSE
			strText:='ORG : Runing ';	
			nInitiStep	:= 17;
		END_IF;	
	//Axis Find Home
	16:
		MC_Home.Execute:=TRUE;
		IF MC_Home.Done THEN
			nInitiStep	:= 17;
		END_IF
		
	
	//Axis Go Abs SDANDBY Pos
	17:
		MC_MoveAbsolute(Axis:= Axis_BoxPullOut,Execute:=TRUE,Position:= RunParameter.Unboxing_PullOut,Velocity:= RunParameter.Unboxing_Velo);
			
		IF MC_MoveAbsolute.Done THEN
			MC_Home(Axis:= Axis_BoxPullOut,Execute:=FALSE);
			MC_MoveAbsolute(Axis:= Axis_BoxPullOut,Execute:=FALSE);	
			nInitiStep	:= 20;
		END_IF	
		
		
		
	//JobDone		
	20:
		strText:='ORG : Done ';
		Initialization	:= TRUE;	
	//Error step
	99:	
		IF Axis_BoxPullOut.DeviceErrorcode <> 0  THEN
			EventLogger.eEventType	:= E_EventType.Error;
			EventLogger.strEventText:= 'UnboxServo Driver Error';
			EventLogger.strEventText:= CONCAT(EventLogger.strEventText,WORD_TO_STRING(Axis_BoxPullOut.DeviceErrorcode));
			EventLogger();
		END_IF
		
		nInitiStep	:= 100;
END_CASE
END_METHOD

{warning 'add property implementation'}
PROPERTY NoEntry : BOOL
GET
END_GET
END_PROPERTY

{warning 'add method implementation '}
METHOD Pause : BOOL
END_METHOD

METHOD Process : BOOL		//OOP Return
VAR_INPUT
	bHlatMode	: BOOL;		//OOP Var
END_VAR
VAR
	_strTemp	:STRING[50];
END_VAR
_bProcessScan	:= TRUE;
//判斷 

IF _bError THEN
	strText	:= 'OpenBox:Error ';
	strText	:= CONCAT(Status,INT_TO_STRING(nStep));
END_IF;
//半自動模式
IF NOT bHlatMode  THEN
	nStep:= nNextStep;	
END_IF;

_bHaltPause	:= nStep<> nNextStep;
IF _bError OR _bHaltPause THEN
	RETURN;
END_IF

//主程序 
IF NOT _bHaltPause THEN
	tmrloadIn(in:= NOT tmrloadIn.q , PT:=RunParameter.Unboxing_DelayTime[0]);	
	IF tmrloadIn.Q THEN
		IF NOT Sen_BoxsideFeed THEN
			wPunchcounter	:= 	wPunchcounter + 1 ;
			Cyl_BoxSidePitch.qExtendCoil:= TRUE;
			ELSE
			wPunchcounter	:= 0;			
		END_IF
	END_IF;
	tmrloadIn2(IN:= Cyl_BoxSidePitch.iEndSensor ,PT:= T#1S);
	IF tmrloadIn2.q THEN
		Cyl_BoxSidePitch.qExtendCoil:= FALSE;			
	END_IF
	
	
	CASE nStep OF
		0:
			tmrDelay(IN:=FALSE);
			MC_MoveAbsolute(Axis:=Axis_BoxPullOut,Execute:=FALSE);
			IF Axis_BoxPullOut.Status.MotionState= MC_AXISSTATE_STANDSTILL AND Axis_BoxPullOut.Status.Homed THEN
				strText:= '';
				nNextStep	:= 10;
				nStep		:= 10;
				ELSE
				nNextStep	:= 100;
				nStep		:= 100;	
				strText:= '馬達狀態異常 ';			
			END_IF;
			
		10:
			MC_MoveAbsolute(Axis:= Axis_BoxPullOut,Execute:=TRUE,Position:= RunParameter.Unboxing_PullOut,Velocity:= RunParameter.Unboxing_Velo);
			IF MC_MoveAbsolute.Done THEN
				MC_MoveAbsolute(Axis:=Axis_BoxPullOut,Execute:=FALSE);
				nNextStep	:= 15;
			END_IF	
		15:
			Cyl_AxisBoxCatch.qExtendCoil	:= TRUE;
			IF Cyl_AxisBoxCatch.iEndSensor THEN
				nNextStep	:= 20;
			END_IF
		20:
			Vacm_AxisCatchBox:= TRUE;
			IF Sen_AxisBoxCatchVacumm THEN
				nNextStep	:= 21;
			END_IF
		21:
			Cyl_AxisBoxCatch.qExtendCoil	:= FALSE;	
			IF Cyl_AxisBoxCatch.iOriginSensor THEN
				nNextStep	:= 22;
			END_IF			
		22:
			Cyl_Axis90.qExtendCoil	:= TRUE;	
			tmrDelay(IN:= Cyl_Axis90.iEndSensor , pt:= T#1S);
			IF Cyl_Axis90.iEndSensor THEN
				tmrDelay(IN:=FALSE);
				nNextStep	:= 23;
			END_IF
		23:		
			Vacm_Axis90				:= TRUE;
			IF Sen_Axis90Vacumm THEN
				nNextStep	:= 24;
			END_IF
		24:
			Cyl_AxisBottom.qExtendCoil	:= TRUE;
			IF Cyl_AxisBottom.iEndSensor THEN
				nNextStep	:= 25;
			END_IF

		25:
			MC_MoveAbsolute(Axis:= Axis_BoxPullOut,Execute:=TRUE,Position:= RunParameter.Unboxing_PullOut+60,Velocity:= RunParameter.Unboxing_Velo);


			IF MC_MoveAbsolute.Done THEN
				MC_MoveAbsolute(Axis:=Axis_BoxPullOut,Execute:=FALSE);
				nNextStep	:= 26;
			END_IF
		26:
			Cyl_BeltBottom.qExtendCoil	:= TRUE;
			IF  Cyl_BeltBottom.iEndSensor THEN
				nNextStep	:= 27;
			END_IF		

		27:
			Cyl_BoxSideBottom.qExtendCoil	:= TRUE;
			IF Cyl_BoxSideBottom.iEndSensor THEN
				nNextStep	:= 28;
			END_IF

		28:
			tmrDelay(IN:=FALSE);
			strText:= 'Wait for Next St. ';	

			IF M_Sealing2.Connect = 'OpenBox In' THEN
				nNextStep	:= 30;
			END_IF
			
			IF NOT OP.xAutoMode THEN
				nNextStep	:= 30;
			END_IF
	
		30:
			//MC_MoveAbsolute(Axis:= Axis_BoxPullOut,Execute:=TRUE,Position:= RunParameter.Unboxing_LoadOut,Velocity:= RunParameter.Unboxing_Velo);
			MC_MoveAbsolute(Axis:= Axis_BoxPullOut,Execute:=TRUE,Position:= RunParameter.Unboxing_LoadOut,Velocity:= 100);

		IF Sen_BeltLoadIn THEN
				Cyl_BeltBottom.qExtendCoil		:= TRUE;
				Cyl_BoxSideBottom.qExtendCoil	:= FALSE;
				Vacm_AxisCatchBox				:=FALSE;
				//Cyl_AxisBottom.qExtendCoil		:= FALSE;
				Cyl_BeltBottom.qExtendCoil		:= FALSE;
				//Cyl_Axis90.qExtendCoil			:= FALSE;	
				Vacm_Axis90						:= FALSE;
			END_IF
			tmrDelay(IN:=MC_MoveAbsolute.Done,PT:=T#2S);
			IF tmrDelay.Q  THEN
				Cyl_BoxSideBottom.qExtendCoil	:= FALSE;
				Vacm_AxisCatchBox			:=FALSE;
				Cyl_AxisBottom.qExtendCoil	:= FALSE;
				Cyl_AxisBottom.qExtendCoil	:= FALSE;
				Cyl_BeltBottom.qExtendCoil	:= FALSE;
				Cyl_Axis90.qExtendCoil	:= FALSE;	
				Vacm_Axis90				:= FALSE;
				MC_MoveAbsolute(Axis:=Axis_BoxPullOut,Execute:=FALSE);
				nNextStep	:= 50;
			END_IF		

	

		50:
			IF OP.xAutoMode AND M_Sealing2.Connect = 'OpenBox In' THEN
				nNextStep	:= 0;
			END_IF
			;
	END_CASE
END_IF;

Process	:= nStep =50;
END_METHOD

PROPERTY Status : STRING(50)
GET
END_GET
END_PROPERTY

END_FUNCTION_BLOCK

// ---- 02_Unit/01_Customization/Ass_LoadPic.TcPOU
FUNCTION_BLOCK Ass_LoadPic IMPLEMENTS ITF_AutoStructCommand
VAR_INPUT
END_VAR
VAR_OUTPUT
END_VAR
VAR
	strText	:STRING;
	i	:INT;
	_bProcessScan,_bInitialScan		: BOOL;
	_bHalt , _bError,_bHaltPause	: BOOL;
	nStep,nInitiStep ,nNextStep 	: INT;
	fbHomeInside,fbHomeOutside		: MC_Home;
	fbMC_GearIn						: MC_GearIn;
	fbMC_GearOut					: MC_GearOut;
	fbMC_AbsLoad1,fbMC_AbsLoad2		: MC_MoveAbsolute;
	fbMC_Mode1	,fbMC_Mode2			:MC_MoveModulo;
	fbMC_INC1,fbMC_INC2	:MC_MoveRelative;
	_tmrT0,tmrStopper							: TON;
	temp:DWORD;
	bReady: BOOL;
END_VAR

IF NOT _bInitialScan AND NOT _bProcessScan  THEN
	fbHomeInside.Execute:=FALSE;
	fbHomeOutside.Execute:=FALSE;
END_IF


IF NOT _bInitialScan THEN
	nInitiStep	:= 0;
END_IF

_bInitialScan:=FALSE;



IF NOT _bProcessScan THEN
	nNextStep	:= 0;
	nStep		:= 0;
END_IF

_bProcessScan	:=FALSE;






fbHomeInside(Axis:= Axis_load1,Position:= Setting_Unload1_ORG_Offset*-1,bCalibrationCam:= NOT Sen_AxisLoad1ORG);
fbHomeOutside(Axis:= Axis_load2,Position:= Setting_Unload2_ORG_Offset*-1,bCalibrationCam:= NOT Sen_AxisLoad2ORG);

METHOD _Clearfb : BOOL
VAR_INPUT
END_VAR
	fbMC_GearIn(Master:=Axis_load1,Slave:=Axis_load2,Execute:=FALSE);
	fbMC_GearOut(Slave:=Axis_load2,Execute:=FALSE);
	fbHomeInside(Axis:= Axis_load1,bCalibrationCam:= FALSE,Execute:=FALSE);
	fbHomeOutside(Axis:= Axis_load2,bCalibrationCam:= FALSE,Execute:=FALSE);
	_tmrT0(IN:=FALSE);
	nInitiStep:=0;
END_METHOD

{warning 'add property implementation'}
PROPERTY Connect : STRING(50)
GET
CASE nStep OF
 10:
	Connect	:= 'Seal In';
20:
	Connect	:= 'LoadIng';
 25:
	Connect	:= 'Seal In';	
	ELSE	
	Connect	:= '';		
END_CASE
END_GET
SET
END_SET
END_PROPERTY

PROPERTY Error : BOOL
GET
Error := _bError;
END_GET
END_PROPERTY

METHOD ErrorClear : BOOL
_bError	:= FALSE;
END_METHOD

{warning 'add method implementation '}
METHOD FB_init : BOOL
VAR_INPUT
	(* if TRUE, the retain variables are initialized (warm start / cold start)*)
	bInitRetains	: BOOL;
	(* if TRUE, the instance afterwards gets moved into the copy code (online change)*)
	bInCopyCode	: BOOL;
END_VAR
END_METHOD

{warning 'add method implementation '}
METHOD HaltStepContiune : BOOL
END_METHOD

METHOD Initialization : BOOL
VAR_INPUT
	_Testmode	:BOOL;
END_VAR
VAR
	bConfig: BOOL;
END_VAR
_bInitialScan	:= TRUE;

CASE nInitiStep OF
	0:
		RB_CS_PickIO.cmd_bBoxInPos	:=FALSE;
		fbMC_AbsLoad1(Axis:= Axis_load1,Velocity:= 100,Execute:= FALSE);
		fbMC_AbsLoad2(Axis:= Axis_load2,Velocity:= 100,Execute:= FALSE);
		fbHomeInside.Execute:=FALSE;
		fbHomeOutside.Execute:=FALSE;
		fbMC_GearOut(Slave:= Axis_load2,Execute:=FALSE);
		_tmrT0(IN:=FALSE);
		Cyl_UnloadDef.qExtendCoil	:= FALSE;
		strText:='ORG : Initial ';
		IF AssRoller.Initialization() THEN
			nInitiStep := 1;
		END_IF
	1:
		_tmrT0(IN:= NOT _tmrT0.Q ,PT:= T#1S);
		CASE Axis_load1.Status.MotionState OF
			MC_AXISSTATE_DISABLED:
			 	Axis_load1.ServoOn();
			MC_AXISSTATE_ERRORSTOP:
				Axis_load1.Reset();
			MC_AXISSTATE_STOPPING:
				Axis_load1.Stop();
			MC_AXISSTATE_SYNCHRONIZEDMOTION:
			;
		END_CASE;		
		CASE Axis_load2.Status.MotionState OF
			MC_AXISSTATE_DISABLED:
			 	Axis_load2.ServoOn();
			MC_AXISSTATE_ERRORSTOP:
				Axis_load2.Reset();
			MC_AXISSTATE_STOPPING:
				Axis_load2.Stop();
			MC_AXISSTATE_SYNCHRONIZEDMOTION:
				fbMC_GearOut(Slave:= Axis_load2,Execute:=TRUE);
		END_CASE;			
		
		IF  Axis_load1.Status.MotionState=MC_AXISSTATE_STANDSTILL AND Axis_load2.Status.MotionState=MC_AXISSTATE_STANDSTILL THEN
			_tmrT0(IN:=FALSE);
			nInitiStep	:=5 ;
		END_IF
		IF _tmrT0.Q THEN
			_tmrT0(IN:=FALSE);
			nInitiStep	:= 5;		
		END_IF
	5:
		bConfig			:=TRUE;
		IF NOT Axis_load1.Status.StandStill THEN
			bConfig			:=FALSE;
			EventLogger.eEventType		:= 4;
			EventLogger.strEventText	:= 'RightAxis Error ';	
			EventLogger();					
		END_IF
		IF NOT Axis_load2.Status.StandStill THEN
			bConfig			:=FALSE;
			EventLogger.eEventType		:= 4;
			EventLogger.strEventText	:= 'LefthtAxis Error';	
			EventLogger();					
		END_IF
		
		IF bConfig THEN
			IF NOT OP.xAutoMode THEN
				EventLogger.eEventType		:= 2;
				EventLogger.strEventText	:= 'LoadIn servo ORG Runing ';	
				EventLogger();
			END_IF;
			_tmrT0(IN:= FALSE);
			nInitiStep:= 10 ;
			strText:='ORG : Runing ';
			ELSE
			EventLogger.eEventType		:= 4;
			EventLogger.strEventText	:= 'Exceptions Cause interruptions!! ';	
			EventLogger();
			OP.xAutoRuning	:=FALSE;
			nInitiStep := nInitiStep +100;	
			strText:='ORG : Failed  ';
		END_IF			
		
	10:
		fbHomeInside.Execute:=TRUE;
		fbHomeOutside.Execute:=TRUE;
		fbMC_AbsLoad1(Axis:= Axis_load1,Position:= 0,Velocity:= RunParameter.Load_Velo,Execute:= fbHomeInside.Done );
		fbMC_AbsLoad2(Axis:= Axis_load2,Position:= 0,Velocity:= RunParameter.Load_Velo,Execute:=  fbHomeOutside.Done);
	
		IF fbMC_AbsLoad1.Done AND fbMC_AbsLoad2.Done THEN
			fbHomeInside.Execute:=FALSE;
			fbHomeOutside.Execute:=FALSE;
			fbMC_AbsLoad1(Axis:= Axis_load1,Velocity:= RunParameter.Load_Velo,Execute:=FALSE );
			fbMC_AbsLoad2(Axis:= Axis_load2,Velocity:= RunParameter.Load_Velo,Execute:=FALSE );
			strText:='ORG : Done ';
			nInitiStep	:= 20 ;
		END_IF
	20:
		Initialization := TRUE;

END_CASE;
END_METHOD

{warning 'add property implementation'}
PROPERTY NoEntry : BOOL
GET
END_GET
END_PROPERTY

{warning 'add method implementation '}
METHOD Pause : BOOL
END_METHOD

METHOD Process : BOOL
VAR_INPUT
	bHlatMode	: BOOL;
END_VAR
_bProcessScan	:= TRUE;
//判斷 

IF _bError THEN
	strText	:= 'OpenBox:Error ';
	strText	:= CONCAT(Status,INT_TO_STRING(nStep));
END_IF;
//半自動模式
IF NOT bHlatMode  THEN
	nStep:= nNextStep;	
END_IF;

_bHaltPause	:= nStep<> nNextStep;
IF _bError OR _bHaltPause THEN
	RETURN;
END_IF
fbMC_INC1(Axis:= Axis_load1,Distance:= 1005,Velocity:= RunParameter.Load_Velo);
fbMC_INC2(Axis:= Axis_load2,Distance:= 1005,Velocity:= RunParameter.Load_Velo);
fbMC_Mode1(Axis:= Axis_load1,Velocity:= fbMC_AbsLoad1.Velocity,Direction:= MC_Positive_Direction);
fbMC_Mode2(Axis:= Axis_load2,Velocity:= fbMC_AbsLoad1.Velocity,Direction:= MC_Positive_Direction);
fbMC_AbsLoad1(Axis:= Axis_load1,Position:= RunParameter.Load_RBLoadin,Velocity:= RunParameter.Load_Velo);
fbMC_AbsLoad2(Axis:= Axis_load2,Position:= RunParameter.Load_RBLoadin,Velocity:= RunParameter.Load_Velo);	

//主程序 
IF NOT _bHaltPause THEN
	CASE nStep OF
		0:
			fbMC_AbsLoad1.Execute:=FALSE;
			fbMC_AbsLoad2.Execute:=FALSE;
			fbMC_INC1.Execute:=FALSE;
			fbMC_INC2.Execute:= FALSE;
			fbMC_Mode1.Execute:= FALSE;
			fbMC_Mode2.Execute:= FALSE;
			fbHomeInside(Axis:= Axis_load1,Execute:=FALSE);
			fbHomeOutside(Axis:= Axis_load2,Execute:=FALSE);
			_tmrT0(IN:=FALSE);			
			nNextStep:= 5;
		
		5:
			fbMC_AbsLoad1(Axis:= Axis_load1,Position:= 0,Velocity:= RunParameter.Load_Velo,Execute:= TRUE);
			fbMC_AbsLoad2(Axis:= Axis_load2,Position:= 0,Velocity:= RunParameter.Load_Velo,Execute:= TRUE);		
			IF fbMC_AbsLoad1.Done AND fbMC_AbsLoad2.Done THEN
				fbMC_AbsLoad1(Axis:= Axis_load1,Velocity:= RunParameter.Load_Velo,Execute:=FALSE );
				fbMC_AbsLoad2(Axis:= Axis_load2,Velocity:= RunParameter.Load_Velo,Execute:=FALSE );
				nNextStep	:= 10 ;
			END_IF		
		10:
			IF OP.xAutoMode THEN
				IF M_Sealing2.Connect='LoadPic In' THEN	
					nNextStep	:= 11 ;
				END_IF;
			END_IF
			
			IF NOT OP.xAutoMode THEN
				IF Sen_BeltLoadOut THEN
					nNextStep	:= 11 ;
				END_IF;			
			END_IF

		11:
			_tmrT0(IN:= NOT Sen_BeltLoadOut ,pt:= T#0.5S);
			IF _tmrT0.Q THEN
				_tmrT0(IN:=FALSE);
				nNextStep	:= 15 ;
			END_IF
			
		15:
			Cyl_UnloadDef.qExtendCoil	:= TRUE;
			fbMC_Mode1.Execute:= TRUE;
			fbMC_Mode1.Position	:= Parameter_PERSISTENT.RunParameter.Load_RBLoadin;
			fbMC_Mode2.Execute:= TRUE;
			fbMC_Mode2.Position	:= Parameter_PERSISTENT.RunParameter.Load_RBLoadin;	
			IF fbMC_Mode1.Done AND fbMC_Mode2.Done THEN
				fbMC_Mode1.Execute:= FALSE;
				fbMC_Mode2.Execute:= FALSE;	
				nNextStep	:= 16 ;			
			END_IF


	
		16:
			IF Cyl_UnloadDef.iEndSensor  THEN
				nNextStep	:= 20 ;
			END_IF	
			
		20:	// 允許手臂loadin
			IF RB_CS.LoadingDone() THEN
				bReady	:= M_Sealing2.Connect = 'Ready';
				_tmrT0(IN:=FALSE);
				nNextStep	:= 25 ;
			END_IF	
		25:
			Cyl_UnloadDef.qExtendCoil	:= FALSE;
			IF Roller_LoadcellUD.iLowPos AND Cyl_UnloadDef.iOriginSensor THEN
				IF bReady THEN
					nNextStep	:= 30 ;
					ELSE
					nNextStep	:= 31 ;
				END_IF;	
			END_IF
		30:	
			tmrStopper(IN:= NOT Sen_UnloadLoadPos ,PT := T#0.5S);
			IF tmrStopper.q THEN
				Cyl_UnloadDef.qExtendCoil	:= TRUE;
			END_IF
			fbMC_INC1.Execute:= TRUE;
			fbMC_INC2.Execute:= TRUE;	
			IF fbMC_INC2.Done AND fbMC_INC1.Done THEN
				fbMC_INC1.Execute:= FALSE;
				fbMC_INC2.Execute:= FALSE;	
				bReady	:=FALSE;
				Cyl_UnloadDef.qExtendCoil	:= TRUE;
				tmrStopper(IN:=FALSE);
				nNextStep	:= 16 ;
			END_IF;
		31:	
			fbMC_Mode1.Execute:= TRUE;
			fbMC_Mode1.Position	:= 0;
			fbMC_Mode2.Execute:= TRUE;
			fbMC_Mode2.Position	:= 0;	
			IF fbMC_Mode1.Done AND fbMC_Mode2.Done THEN
				fbMC_Mode1.Execute:= FALSE;
				fbMC_Mode2.Execute:= FALSE;	
				nNextStep	:= 10 ;			
			END_IF
			
			(*
			IF Initialization(FALSE) THEN
				nNextStep	:= 0 ;
				IF bReady THEN
					nNextStep	:= 15 ;
				END_IF
			END_IF
		*)
		
			
		
	END_CASE;
END_IF;
		
Process	:= nStep =50;
END_METHOD

PROPERTY Status : STRING(50)
GET
END_GET
END_PROPERTY

END_FUNCTION_BLOCK

// ---- 02_Unit/01_Customization/Ass_RBStack.TcPOU
FUNCTION_BLOCK Ass_RBStack IMPLEMENTS ITF_AutoStructCommand
VAR_INPUT
END_VAR
VAR_OUTPUT
END_VAR
VAR
	strText	:STRING;
	i,_CaptureStep	:INT;
	_bProcessScan,_bInitialScan: BOOL;
	_bHalt , _bError,_bHaltPause: BOOL;
	nStep,nInitiStep ,nNGStep,nShackStep,nPalletStep	: INT;
	_tmrT0,_tmrT1,tmrshock	,tmrNG,tmrPalletTime,tmrAutoPass,tmrStarRetry		:TON;
	bBoxPass: BOOL;
	nNextStep: INT;
	rPalletInPos	:Tc2_Standard.R_TRIG;
	PalletNumb,PalletSensorNumb,Palletslot			:INT;
	bAutoPass: BOOL;
	wRetry:INT;
END_VAR

IF NOT _bInitialScan THEN
	nInitiStep	:= 0;
END_IF

_bInitialScan:=FALSE;



IF NOT _bProcessScan THEN
	nNextStep	:= 0;
	nStep		:= 0;
END_IF

_bProcessScan	:=FALSE;

//
rPalletInPos(CLK:= RB_KR_StackingIO.fb_bPalletInPos);
IF rPalletInPos.Q THEN
	PalletSensorNumb:= PalletSensorNumb + 1;
END_IF

CASE nPalletStep OF
	0://
		IF RB_KR_StackingIO.fb_bPalletInPos THEN
			Palletslot	:= 0;
			RB_KR_StackingIO.cmd_wLayer_No	:= INT_TO_BYTE(RunParameter.StackingRB_LayerData[0]);
			PalletNumb	:= PalletSensorNumb	;
			nPalletStep:= 5;
		END_IF

	5://
		Hmi_bChangePalletDemand	:= FALSE;
		RB_KR_StackingIO.cmd_bPallet_AllowPut	:= RB_KR_StackingIO.fb_bPalletInPos ;
				
		IF  RB_KR_StackingIO.fb_bPalletFinish THEN
			DoNotLoadingRB	:= TRUE;
			nPalletStep:= 10;
			RB_KR_StackingIO.cmd_bPallet_AllowPut	:= FALSE;
			PalletNumb	:= PalletSensorNumb	;
			Counter_Pallet	:= Counter_Pallet + 1;
			Palletslot		:= Palletslot + 1;
			//check pallet Safe
			IF RunParameter.StackingRB_LayerData[Palletslot] =0 THEN
				Palletslot	:= 0;
			END_IF
		END_IF
	10:

		RB_KR_StackingIO.cmd_bCount0	:= TRUE;
		IF RB_KR_StackingIO.fb_wPartNo = 1 AND NOT RB_KR_StackingIO.fb_bPalletFinish THEN
			RB_KR_StackingIO.cmd_bCount0	:= FALSE;
			nPalletStep:= 15;
		END_IF	
	15://偵測換版 
		
		Hmi_bChangePalletDemand	:= TRUE;
		IF Hmi_bAutoChangePallet THEN
			tmrPalletTime(IN:= RB_KR_StackingIO.fb_bPalletInPos AND PalletNumb <> PalletSensorNumb );
			IF tmrPalletTime.Q THEN
				PalletNumb	:= PalletSensorNumb	;
				RB_KR_StackingIO.cmd_wLayer_No	:= INT_TO_BYTE(RunParameter.StackingRB_LayerData[Palletslot]);
				nPalletStep:= 5;
			END_IF
		END_IF
		IF Hmi_bChangePalletbtn THEN
			PalletNumb	:= PalletSensorNumb	;
			RB_KR_StackingIO.cmd_wLayer_No	:= INT_TO_BYTE(RunParameter.StackingRB_LayerData[Palletslot]);
			nPalletStep:= 5;			
			Hmi_bChangePalletbtn:=FALSE;
		END_IF

END_CASE

{warning 'add property implementation'}
PROPERTY Connect : STRING(50)
GET
END_GET
SET
END_SET
END_PROPERTY

{warning 'add property implementation'}
PROPERTY Error : BOOL
GET
END_GET
END_PROPERTY

{warning 'add method implementation '}
METHOD ErrorClear : BOOL
END_METHOD

{warning 'add method implementation '}
METHOD FB_init : BOOL
VAR_INPUT
	(* if TRUE, the retain variables are initialized (warm start / cold start)*)
	bInitRetains	: BOOL;
	(* if TRUE, the instance afterwards gets moved into the copy code (online change)*)
	bInCopyCode	: BOOL;
END_VAR
END_METHOD

{warning 'add method implementation '}
METHOD HaltStepContiune : BOOL
END_METHOD

METHOD Initialization : BOOL
VAR_INPUT
	_Testmode	: BOOL;
END_VAR
_bInitialScan:=TRUE;

CASE nInitiStep OF
	0:		
		strText					:= 'ORG : Inital';
		Cyl_ExitStopper.qExtendCoil	:=FALSE;
		Cyl_ExitClip.qExtendCoil	:=FALSE;
		Roller_Exit.qRun			:=FALSE;	
		nInitiStep				:= 5;	
	5:
		IF 	NOT Sen_ExitLoadIn AND NOT Sen_ExitBoxCheck AND NOT Sen_ExitComvStop THEN
			nInitiStep				:= 10;	
		END_IF;
	10:
			strText:='ORG : Done ';
			Initialization	:= TRUE;
	
END_CASE;
END_METHOD

{warning 'add property implementation'}
PROPERTY NoEntry : BOOL
GET
END_GET
END_PROPERTY

{warning 'add method implementation '}
METHOD Pause : BOOL
END_METHOD

METHOD Process : BOOL
VAR_INPUT
	bHlatMode	: BOOL;
END_VAR
_bProcessScan:=TRUE;


CASE nStep OF
	0:	
		Bundling_yPause			:=FALSE;
		_tmrT0(IN:=FALSE);
		_tmrT1(IN:=FALSE);
		_CaptureStep				:= 0;
		Roller_Exit.qRun			:= TRUE;
		Cyl_ExitStopper.qExtendCoil	:=FALSE;
		IF Sen_ExitLoadIn THEN
			nStep	:= 5;
		END_IF
		IF bAutoPass	THEN
			nStep	:= 11;
		END_IF
		
	5:
		_tmrT0(IN:=Sen_ExitBoxCheck,PT:=T#0.2S);
		IF _tmrT0.Q THEN
			Cyl_ExitStopper.qExtendCoil:=	TRUE;
			_tmrT0(IN:=FALSE);
			Roller_Exit.qRun			:= FALSE;
			Cyl_ExitClip.qExtendCoil	:= TRUE;
			nStep	:= 10;
		END_IF
	10:
		_tmrT0(IN:=TRUE,PT:=T#0.2S);	
		_tmrT1(IN:=Sen_ExitComvStop,PT:=T#0.2S);		
		IF _tmrT0.Q THEN
			IF _tmrT1.q THEN
				_tmrT0(IN:=FALSE);
				_tmrT1(IN:=FALSE);
				Cyl_ExitClip.qExtendCoil	:= FALSE;
				IF HardwareIO.RB_KR_SysIO.iCONTROL_READY THEN
				nStep	:= 15;
				ELSE
				nStep	:= 20;	
			END_IF;
			END_IF;		
		END_IF
	11:
		tmrAutoPass(IN:= TRUE,PT:=T#2S);
		IF tmrAutoPass.Q THEN
			tmrAutoPass(IN:= FALSE);
			nStep	:= 15;
		END_IF
	15://通知手臂
		IF Sen_ExitLoadIn THEN
			Bundling_yPause			:=TRUE;
		END_IF;
		tmrStarRetry(IN:=NOT tmrStarRetry.Q  ,PT:=T#0.5S);
		IF tmrStarRetry.Q THEN
			IF RB_KR_SysIO.iEXT_CONTROL AND NOT DoNotLoadingRB THEN
				IF RB_KR_SysIO.iPGNO_REQ THEN
					tmrStarRetry.IN := TRUE;
					RB_KR_SysIO.qEXT_START:= TRUE;
				END_IF
				IF NOT RB_KR_SysIO.iPGNO_REQ AND NOT RB_KR_SysIO.iRobotRunning THEN
					tmrStarRetry.IN 	:= TRUE;
					RB_KR_SysIO.qEXT_START:= TRUE;
				END_IF		
			END_IF;	
		END_IF
		

		
		CASE _CaptureStep OF	
		0:
			RB_KR_StackingIO.cmd_bPartInPos	:= TRUE;
			_CaptureStep	:= 5;
			
		5:
			IF RB_KR_StackingIO.fb_bPickFinish THEN
				RB_KR_StackingIO.cmd_bPartInPos	:= FALSE;
				_CaptureStep	:= 10;
			END_IF
	
		10:
			IF NOT RB_KR_StackingIO.fb_bPickFinish THEN
				_CaptureStep	:= 15;
			END_IF		
		15:
			_CaptureStep	:= 0;
			nStep			:= 20;
		END_CASE;	

		
	20:
		IF Sen_ExitLoadIn THEN
			Bundling_yPause			:=TRUE;
		END_IF;
		IF NOT Sen_ExitLoadIn AND NOT Sen_ExitBoxCheck AND NOT Sen_ExitComvStop THEN
			nStep	:= 0;
		END_IF
	
	
	
	

END_CASE
END_METHOD

METHOD ResetPallet : BOOL
VAR_INPUT
END_VAR
nPalletStep	:= 0;
END_METHOD

{warning 'add property implementation'}
PROPERTY Status : STRING(50)
GET
END_GET
END_PROPERTY

END_FUNCTION_BLOCK

// ---- 02_Unit/01_Customization/FB_RollRightAngle.TcPOU
FUNCTION_BLOCK FB_RollRightAngle
VAR_INPUT
	ref_Roller 	:REFERENCE TO ST_Inventer;
	ref_Belt 	:REFERENCE TO ST_Inventer;
	ref_UD 		:REFERENCE TO ST_InventerUD;
END_VAR
VAR_OUTPUT
	o_bError :BOOL;
END_VAR
VAR
	_Belt	:BOOL;
	ldfBeltOff	:F_TRIG;
	
	_Roller	:BOOL;
	tmrRollerDelay	:TON;
	ldfRollerOff	:F_TRIG;
	
	tmrErrorDelay	:TON;
END_VAR

//Error cont.
o_bError := ref_Belt.iError	OR ref_Roller.iError OR ref_UD.iError OR  tmrErrorDelay.Q;





//皮帶
ldfBeltOff(CLK:=_Belt);
IF ldfBeltOff.q THEN
	tmrErrorDelay(IN:=FALSE);
	ref_Belt.qRun	:=FALSE;
	ref_UD.qSign	:= FALSE;
	ref_UD.qRun		:= FALSE;
END_IF
_Belt	:=FALSE;


//進入滾珠
ldfRollerOff(CLK:=_Roller);

IF ldfRollerOff.Q THEN
	tmrErrorDelay(IN:=FALSE);
	tmrRollerDelay(IN:=FALSE);
	ref_Roller.qRun	:=FALSE;
	ref_UD.qSign	:= FALSE;
	ref_UD.qRun		:= FALSE;
END_IF

_Roller	:=FALSE;

METHOD Belt : BOOL
VAR_INPUT
END_VAR
_Belt	:= TRUE;
ref_Belt.qRun	:= TRUE;
//Error Timer 
tmrErrorDelay(IN:=NOT ref_UD.iHighPos,PT:=T#2S);
//belt In senser Position 
ref_UD.qRun	:= NOT ref_UD.iHighPos;
ref_UD.qSign		:= FALSE;


IF tmrErrorDelay.Q THEN
	ref_UD.qSign	:= FALSE;
	ref_UD.qRun		:= FALSE;
END_IF
END_METHOD

METHOD Initialization : BOOL
VAR_INPUT
END_VAR
_Roller	:= TRUE;
ref_Roller.qRun	:= FALSE;
ref_Belt.qRun	:= FALSE;
//Error Timer 
tmrErrorDelay(IN:=NOT ref_UD.iLowPos,PT:=T#2S);
//
IF NOT ref_UD.iLowPos THEN
	ref_UD.qSign	:= TRUE;
	tmrRollerDelay(IN:=TRUE,PT:= T#20MS);
	ref_UD.qRun	:= tmrRollerDelay.Q ;
	ELSE
	ref_UD.qSign	:= FALSE;
	ref_UD.qRun		:= FALSE;
END_IF

Initialization	:= ref_UD.iLowPos;
END_METHOD

METHOD Roller : BOOL
VAR_INPUT
END_VAR
_Roller	:= TRUE;
ref_Belt.qRun	:= FALSE;
//Error Timer 
tmrErrorDelay(IN:=NOT ref_UD.iLowPos,PT:=T#2S);
//
IF NOT ref_UD.iLowPos THEN
	ref_UD.qSign	:= TRUE;
	tmrRollerDelay(IN:=TRUE,PT:= T#20MS);
	ref_UD.qRun	:= tmrRollerDelay.Q ;
	ELSE
	ref_UD.qSign	:= FALSE;
	ref_UD.qRun		:= FALSE;
	ref_Roller.qRun	:= TRUE	;
END_IF


IF tmrErrorDelay.Q THEN
	ref_UD.qSign	:= FALSE;
	ref_UD.qRun		:= FALSE;
END_IF
END_METHOD

END_FUNCTION_BLOCK

// ---- 02_Unit/99_Other/FB_EL3356_0010.TcPOU
FUNCTION_BLOCK FB_EL3356_0010
VAR_INPUT

	i_tInputFreeze				:TIME:=T#50MS;
	i_rInputFreezeTreshold		:REAL:=10;
END_VAR
VAR_OUTPUT
		(* Status Flag*)
	o_obUnderrange				:BOOL;		//低於範圍
	o_bOverrange				:BOOL;		//超出範圍 
	o_bDataInvalid				:BOOL;		//資料無效 
	o_bError					:BOOL;		//Error
	o_bCalibrationInProgress	:BOOL;		//
	o_bSteadyState				:BOOL;		//穩定中 
	o_bTxPDOToggle				:BOOL;		//刷新資料
	o_bSyncError				:BOOL;		//
	o_rWeight					:REAL;
	strStatus					:STRING(100);
	strSampleMode				:STRING(100);			
END_VAR
VAR
	(* process data OUT*)
	wControl AT %Q*:WORD;
	(* process data IN*)
	wStatus AT %I*:WORD;
	rValue_REAL AT %I*:REAL;
	nValue_Supply AT %I*:DINT;		(*only for voltage measurement, change PDO settings"*)
	nValue_Bridge AT %I*:DINT;		(*only for voltage measurement, change PDO settings"*)
	stEcSlaveAmsNetAdr AT %I*:ST_AmsAddr;
	bWcState AT %I*:BOOL;
	wState AT %I*:WORD;

	
		(* Control commands *)
	bStartManualCalib	:BOOL;		//開始校準	-Control 
	bDisableCalibration	:BOOL;		//停止校準	-Control
	bSampleMode			:BOOL;		//sampleMode	-Control
	bTara				:BOOL;		//去皮		-Control
	//////////
	sEcSlaveAmsNetAdr:T_AmsNetId;
	rValue:REAL;

	fbCoE		:ARRAY [0..10] OF  FB_EcCoESdoWrite;
	wCoeData	:WORD;
	dwCoeData	:DWORD;
	bTermError:BOOL;
	nCntCalibrations:UDINT;
	sfCalibInProgress:R_TRIG;

	_bInitial		,_bSetLoadcell,_bSetRefLoad,_bSetScaleFactor,_bSetZeroCali,_bSetLoadCali ,_bSetCommand,_bTara		:BOOL;
	_Initialbuff	,_SetLoadcell,_SetRefLoad	,_SetScaleFactor,_SetZeroCali,_SetLoadCali	,_SetCommand,_Tara		:WORD;
	

	rValueDiff, rValueL:REAL;
	bActivateAutoInputFreeze:BOOL;
	tofInputFreeze:TOF;
	tInputFreeze:TIME:=T#50MS;
	tTara	:TON := (PT := TIME#500ms);
	sfCntInputFreeze:R_TRIG;
	nCntInputFreeze:UDINT;


END_VAR

	(*example program for EL3356(-0010)
	this demo is designed only for load cell connection, not for 2channel voltage measurement*)

	(*get terminal information*)
o_bOverrange := wStatus.1;
o_bDataInvalid := wStatus.3;
o_bError := wStatus.6;
o_bCalibrationInProgress := wStatus.7;
o_bSteadyState := wStatus.8;
o_bSyncError := wStatus.13;
o_bTxPDOToggle := wStatus.15;
	(*triggers*)
	
//sfZeroCalibration(CLK:=i_bCmd_ZeroCalibration);
//sfFullCalibration(CLK:=i_bCmd_FullCalibration);
//sfTara(CLK:=i_bCmd_Tara);
//sfTaraEEProm(CLK:=i_bCmd_TaraEEProm);
//sfInitial(CLK:= i_bInitial);
//sfWriteLoadcellMaxWeight(CLK:= i_bWriteLoadcellMaxWeight);
//sfbWriteRefWeight(CLK:= i_bWriteRefWeight);


	(*value: Integer or Real value*)
IF (rValue_REAL <> 0) THEN	(*select currently used input data*)
	rValue := rValue_REAL;
	rValue := 0;
END_IF

	(*status*)
IF bWcState THEN
	strStatus := 'Wc fail';
	bTermError := TRUE;
ELSIF NOT (wState.3) THEN
	strStatus := 'Slave not in OP';
	bTermError := TRUE;
ELSIF o_bDataInvalid THEN
	strStatus := 'DataInvalid';
	bTermError := TRUE;
ELSIF o_bError THEN
	strStatus := 'Channel Error';
	bTermError := TRUE;
ELSIF o_bOverrange THEN
	strStatus := 'Overrange';
	bTermError := TRUE;
ELSE
	strStatus := 'ok';
	bTermError := FALSE;
END_IF

	(*sample mode 0/1*)
strSampleMode := SEL(bSampleMode, '0', '1');

	(*count calibrations*)
sfCalibInProgress(CLK:= o_bCalibrationInProgress, Q=> );
nCntCalibrations := SEL(sfCalibInProgress.Q , nCntCalibrations, nCntCalibrations+ 1);

	(*Coe parameter administration*)
sEcSlaveAmsNetAdr := F_CreateAmsNetId(nIds:=stEcSlaveAmsNetAdr.netId );

	(*test input freeze
this lines are for a small demonstration of Input freeze: when difference of loadvalue, compared to last PLC cycle, is over rInputFreezeTreshold
then InputFreeze is activated by tofInputFreeze for some time. See screenshot in documentation for further explanations*)
rValueDiff := rValue - rValueL;
rValueL := rValue;
tofInputFreeze(IN:= bActivateAutoInputFreeze AND (ABS(rValueDiff) >i_rInputFreezeTreshold) , PT:= tInputFreeze, Q=> , ET=> );
sfCntInputFreeze(CLK:= tofInputFreeze.Q , Q=> );
nCntInputFreeze := SEL(sfCntInputFreeze.Q , nCntInputFreeze, nCntInputFreeze+ 1);

(*++++++++++++++ CoE communication ++++++++++++++++++++++*)
IF NOT _bInitial THEN
	fbCoE[0](bExecute 	:= FALSE);
	_Initialbuff	:= 0;
END_IF
_bInitial:= FALSE;
//
IF NOT _bSetLoadcell THEN
	fbCoE[1](bExecute 	:= FALSE);
	_SetLoadcell	:= 0;
END_IF
_bSetLoadcell:=FALSE;
//
IF NOT _bSetRefLoad THEN
	fbCoE[2](bExecute 	:= FALSE);
	_SetRefLoad	:= 0;
END_IF
_bSetRefLoad:=FALSE;
//
IF NOT _bSetScaleFactor THEN
	fbCoE[3](bExecute 	:= FALSE);
	_SetScaleFactor	:= 0;
END_IF
_bSetScaleFactor:= FALSE;

//
IF NOT _bSetZeroCali THEN
	fbCoE[4](bExecute 	:= FALSE);
	_SetZeroCali	:= 0;
END_IF
_bSetZeroCali	:= FALSE;
//
IF NOT _bSetLoadCali THEN
	fbCoE[5](bExecute 	:= FALSE);
	_SetLoadCali	:= 0;
END_IF
_bSetLoadCali	:= FALSE;
//
IF NOT _bSetCommand THEN
	fbCoE[6](bExecute 	:= FALSE);
	_SetCommand	:= 0;
END_IF
_bSetCommand	:= FALSE;

//
IF NOT _bTara THEN
	tTara(IN:=FALSE);
	_Tara	:= 0;
	bTara	:= FALSE;
END_IF
_bTara:=FALSE;
	(*output data to terminal*)
wControl.0 := bStartManualCalib;
wControl.1 := bDisableCalibration;
//wControl.2 := i_bInputFreeze OR tofInputFreeze.Q ;
wControl.3 := bSampleMode;
wControl.4 := bTara;

o_rWeight:= rValue_REAL;
//Ext

METHOD GetTara : BOOL
VAR_INPUT
END_VAR
_bTara	:= TRUE;

CASE _Tara OF
	0: 
		bTara	:= TRUE;
		tTara(IN:= TRUE);
		IF tTara.Q THEN
			tTara(IN:= FALSE);
			_Tara	:= 5;
		END_IF

	5:
		GetTara:= TRUE;
END_CASE
END_METHOD

METHOD Initialization : BOOL
VAR_INPUT
END_VAR
//修改CoE object 0x1011:01值为1684107116恢复出厂设置
_bInitial	:= TRUE;

CASE _Initialbuff OF
	0:
		dwCoeData := 1684107116; (* Command zerocalibration*)
		fbCoE[0](
			sNetId		:= sEcSlaveAmsNetAdr,
			nSlaveAddr 	:= stEcSlaveAmsNetAdr.port,
			nSubIndex 	:= 16#01,
			nIndex 		:= 16#1011,
			pSrcBuf 	:= ADR(dwCoeData),
			cbBufLen 	:= SIZEOF(dwCoeData),
			bExecute 	:= TRUE,
			tTimeout 	:= T#5S		
			);
		IF fbCoE[0].bBusy THEN
			_Initialbuff	:= 1;
		END_IF;
			
	1:
		fbCoE[0]();				
		IF NOT fbCoE[0].bBusy THEN
			_Initialbuff	:= 2;
			IF fbCoE[0].bError THEN
				_Initialbuff	:= 5;
			END_IF
		END_IF;	
	2:
		Initialization		:= TRUE;
		fbCoE[0](bExecute 	:= FALSE);
	5:
		Initialization		:= TRUE;
		fbCoE[0](bExecute 	:= FALSE);		
END_CASE
END_METHOD

METHOD SetLoadCalibration : BOOL
VAR_INPUT
END_VAR
_bSetLoadCali	:= TRUE;

CASE _SetLoadCali OF
	0:
		_SetLoadCali	:= 1;
	
	1:
		wCoeData	:= 16#0102;
		fbCoE[5](
			sNetId		:= sEcSlaveAmsNetAdr,
			nSlaveAddr 	:= stEcSlaveAmsNetAdr.port,
			nSubIndex 	:= 16#01,
			nIndex 		:= 16#FB00,
			pSrcBuf 	:= ADR(wCoeData),
			cbBufLen 	:= SIZEOF(wCoeData),
			bExecute 	:= TRUE,
			tTimeout 	:= T#5S		
			);
		IF fbCoE[5].bBusy THEN
			_SetLoadCali	:=2;
		END_IF;
			
	2:
		fbCoE[5]();				
		IF NOT fbCoE[5].bBusy THEN
			_SetLoadCali	:= 3;
			IF fbCoE[5].bError THEN
				_SetLoadCali	:= 5;
			END_IF
		END_IF;	
	3:
		SetLoadCalibration		:= TRUE;
		fbCoE[5](bExecute 	:= FALSE);
	5:

		fbCoE[5](bExecute 	:= FALSE);		
END_CASE
END_METHOD

METHOD SetNomialLoad : BOOL
VAR_INPUT
	MaxWeight:REAL;
END_VAR
//8.	0x8000:24 ("额定值") ，本例的传感器为最大称重1kg，那么就输入1000 
_bSetLoadcell	:= TRUE;

CASE _SetLoadcell OF
	0:
		IF MaxWeight = 0.0 THEN
			_SetLoadcell	:=5;
			ELSE
			_SetLoadcell	:= 1;
		END_IF
	1:
		fbCoE[1](
			sNetId		:= sEcSlaveAmsNetAdr,
			nSlaveAddr 	:= stEcSlaveAmsNetAdr.port,
			nSubIndex 	:= 16#24,
			nIndex 		:= 16#8000,
			pSrcBuf 	:= ADR(MaxWeight),
			cbBufLen 	:= SIZEOF(MaxWeight),
			bExecute 	:= TRUE,
			tTimeout 	:= T#5S		
			);
		IF fbCoE[1].bBusy THEN
			_SetLoadcell	:=2;
		END_IF;
			
	2:
		fbCoE[1]();				
		IF NOT fbCoE[1].bBusy THEN
			_SetLoadcell	:= 3;
			IF fbCoE[1].bError THEN
				_SetLoadcell	:= 5;
			END_IF
		END_IF;	
	3:
		SetNomialLoad		:= TRUE;
		fbCoE[1](bExecute 	:= FALSE);
	5:

		fbCoE[1](bExecute 	:= FALSE);		
END_CASE
END_METHOD

METHOD SetRefLoad : BOOL
VAR_INPUT
	RefLoad:REAL;
END_VAR
//500g的砝码在 0x8000:28 校准负载填写500, (0x8000:24)额定负载填写1000。

_bSetRefLoad	:= TRUE;

CASE _SetRefLoad OF
	0:
		IF RefLoad = 0.0 THEN
			_SetRefLoad	:=5;
			ELSE
			_SetRefLoad	:= 1;
		END_IF
	1:
		fbCoE[2](
			sNetId		:= sEcSlaveAmsNetAdr,
			nSlaveAddr 	:= stEcSlaveAmsNetAdr.port,
			nSubIndex 	:= 16#28,
			nIndex 		:= 16#8000,
			pSrcBuf 	:= ADR(RefLoad),
			cbBufLen 	:= SIZEOF(RefLoad),
			bExecute 	:= TRUE,
			tTimeout 	:= T#5S		
			);
		IF fbCoE[2].bBusy THEN
			_SetRefLoad	:=2;
		END_IF;
			
	2:
		fbCoE[2]();				
		IF NOT fbCoE[2].bBusy THEN
			_SetRefLoad	:= 3;
			IF fbCoE[2].bError THEN
				_SetRefLoad	:= 5;
			END_IF
		END_IF;	
	3:
		SetRefLoad		:= TRUE;
		fbCoE[2](bExecute 	:= FALSE);
	5:

		fbCoE[2](bExecute 	:= FALSE);		
END_CASE
END_METHOD

METHOD SetScaleFactor : BOOL
VAR_INPUT
	ScaleFactor	:REAL;
END_VAR
//0x8000:27 校准负载填写1單位kg , 1000/g

_bSetScaleFactor	:= TRUE;

CASE _SetScaleFactor OF
	0:
		IF ScaleFactor = 0.0 THEN
			_SetScaleFactor	:=5;
			ELSE
			_SetScaleFactor	:= 1;
		END_IF
	1:
		fbCoE[3](
			sNetId		:= sEcSlaveAmsNetAdr,
			nSlaveAddr 	:= stEcSlaveAmsNetAdr.port,
			nSubIndex 	:= 16#27,
			nIndex 		:= 16#8000,
			pSrcBuf 	:= ADR(ScaleFactor),
			cbBufLen 	:= SIZEOF(ScaleFactor),
			bExecute 	:= TRUE,
			tTimeout 	:= T#5S		
			);
		IF fbCoE[3].bBusy THEN
			_SetScaleFactor	:=2;
		END_IF;
			
	2:
		fbCoE[3]();				
		IF NOT fbCoE[3].bBusy THEN
			_SetScaleFactor	:= 3;
			IF fbCoE[3].bError THEN
				_SetScaleFactor	:= 5;
			END_IF
		END_IF;	
	3:
		SetScaleFactor		:= TRUE;
		fbCoE[3](bExecute 	:= FALSE);
	5:

		fbCoE[3](bExecute 	:= FALSE);		
END_CASE
END_METHOD

METHOD SetZeroCalibration : BOOL
VAR_INPUT
END_VAR
_bSetZeroCali	:= TRUE;

//0x8000:27 校准负载填写1單位kg , 1000/g

CASE _SetZeroCali OF
	0:
		_SetZeroCali	:= 1;
	
	1:
		wCoeData	:= 16#0101;
		fbCoE[4](
			sNetId		:= sEcSlaveAmsNetAdr,
			nSlaveAddr 	:= stEcSlaveAmsNetAdr.port,
			nSubIndex 	:= 16#01,
			nIndex 		:= 16#FB00,
			pSrcBuf 	:= ADR(wCoeData),
			cbBufLen 	:= SIZEOF(wCoeData),
			bExecute 	:= TRUE,
			tTimeout 	:= T#5S		
			);
		IF fbCoE[4].bBusy THEN
			_SetZeroCali	:=2;
		END_IF;
			
	2:
		fbCoE[4]();				
		IF NOT fbCoE[4].bBusy THEN
			_SetZeroCali	:= 3;
			IF fbCoE[4].bError THEN
				_SetZeroCali	:= 5;
			END_IF
		END_IF;	
	3:
		SetZeroCalibration		:= TRUE;
		fbCoE[4](bExecute 	:= FALSE);
	5:

		fbCoE[4](bExecute 	:= FALSE);		
END_CASE
END_METHOD

METHOD WriteCommand : BOOL
VAR_INPUT
	wInputData	:WORD;
END_VAR
_bSetCommand	:= TRUE;

CASE _SetCommand OF
	0:
		_SetCommand	:= 1;
	
	1:
		wCoeData	:= wInputData;
		fbCoE[6](
			sNetId		:= sEcSlaveAmsNetAdr,
			nSlaveAddr 	:= stEcSlaveAmsNetAdr.port,
			nSubIndex 	:= 16#01,
			nIndex 		:= 16#FB00,
			pSrcBuf 	:= ADR(wCoeData),
			cbBufLen 	:= SIZEOF(wCoeData),
			bExecute 	:= TRUE,
			tTimeout 	:= T#5S		
			);
		IF fbCoE[6].bBusy THEN
			_SetCommand	:=2;
		END_IF;
			
	2:
		fbCoE[6]();				
		IF NOT fbCoE[6].bBusy THEN
			_SetCommand	:= 3;
			IF fbCoE[6].bError THEN
				_SetCommand	:= 5;
			END_IF
		END_IF;	
	3:
		WriteCommand		:= TRUE;
		fbCoE[6](bExecute 	:= FALSE);
	5:

		fbCoE[6](bExecute 	:= FALSE);		
END_CASE
END_METHOD

END_FUNCTION_BLOCK

// ---- 02_Unit/04_Kuka/RB_KR_PickPlace.TcPOU
FUNCTION_BLOCK RB_KR_PickPlace
VAR_INPUT
	state			AT%I*	:UINT;
	aryEIPInput		AT%I*	:ARRAY [0..63] OF UINT ;
END_VAR
VAR_OUTPUT
	eCSStatus			:E_CS_Status;
	strTextBox			:STRING(50);
	aryEIPOutput		AT%Q*	:ARRAY [0..63] OF UINT ;
	bOffline				:BOOL;
	bBackRun			:BOOL;
END_VAR
VAR
	tmrSimuLoadingDelay,tmrBGRun		:TON;	
	_bLoadingDoneScan	:BOOL;
	tmrSimuPickupDelay,tmrInit	:TON;	
	_bPickUpScan,_bPOUrun,_bInit	:BOOL;
	_POUrun,_PickUpScan		,_LoadingDoneScan,_Init	:INT;	
	tmrPouRun		:TON;
	fbLdf_EnableOff,rPickTrigger	:F_TRIG;
	tmrStartPulse,tmrStopPulse,tmrResetPulse,tmrqPAUSEPulse,tmrCONTINUEPulse,tmrAckPulse	:TON;
	wRetry: INT;
	tPartCycTime:TIME;
	wInitilRetry: INT;
	wBGHistory,wBKtemp	:BYTE;
END_VAR

IO_Mapp();
// =====================================================
// I/O
// =====================================================

fbLdf_EnableOff(CLK:=RB_CS_SysIO.iENABLED);
IF fbLdf_EnableOff.Q THEN
	IF RB_CS_SysIO.qENABLE THEN
		RB_CS_SysIO.qENABLE	:=FALSE;
		EventLogger.eEventType		:= 3;
		EventLogger.strEventText	:= 'RB_CS Enable Off ';	
		EventLogger();
	END_IF
END_IF

tmrStopPulse(IN:= RB_CS_SysIO.qSTOP,PT:=T#0.3S);
IF tmrStopPulse.Q THEN
	RB_CS_SysIO.qSTOP	:=FALSE;
END_IF
tmrStartPulse(IN:= RB_CS_SysIO.qSTART,PT:=T#0.3S);
IF tmrStartPulse.Q THEN
	RB_CS_SysIO.qSTART	:=FALSE;
END_IF
tmrResetPulse(IN:= RB_CS_SysIO.qRESET,PT:=T#0.3S);
IF tmrResetPulse.Q THEN
	RB_CS_SysIO.qRESET	:=FALSE;
END_IF
tmrqPAUSEPulse(IN:= RB_CS_SysIO.qPAUSE,PT:=T#0.3S);
IF tmrqPAUSEPulse.Q THEN
	RB_CS_SysIO.qPAUSE	:=FALSE;
END_IF
tmrCONTINUEPulse(IN:= RB_CS_SysIO.qCONTINUE,PT:=T#0.3S);
IF tmrCONTINUEPulse.Q THEN
	RB_CS_SysIO.qCONTINUE	:=FALSE;
END_IF
tmrAckPulse(IN:= RB_CS_SysIO.qACKNOWLEDGEMSG,PT:=T#0.3S);
IF tmrAckPulse.Q THEN
	RB_CS_SysIO.qACKNOWLEDGEMSG	:=FALSE;
END_IF
rPickTrigger(CLK:= RB_CS_PickIO.cmd_bPartInPos);
IF rPickTrigger.Q THEN
	tPartCycTime:=SF.GetOvertime(0);
END_IF

// =====================================================
// Flag
// =====================================================
IF RB_CS_SysIO.iREADY THEN
	eCSStatus:=E_CS_Status.DriveReady;
	ELSE
	eCSStatus:=E_CS_Status.Idle;	
END_IF


IF RB_CS_SysIO.iENABLED THEN
	eCSStatus:=E_CS_Status.ReadyToWork;	
	IF RB_CS_SysIO.iRUNNING THEN
		eCSStatus:=E_CS_Status.Pou_Runing;	
	END_IF;
	IF RB_CS_SysIO.iPAUSED THEN
		eCSStatus:=E_CS_Status.Pou_Run_Pause;	
	END_IF;	
	IF RB_CS_SysIO.iSTOPPED THEN
		eCSStatus:=E_CS_Status.Pou_Run_Down;	
	END_IF
END_IF

IF RB_CS_SysIO.iERROR  THEN
	eCSStatus:=E_CS_Status.Error;	
END_IF

IF RB_CS_SysIO.iESTOP_ON THEN
	RB_CS_SysIO.qENABLE	:=FALSE;
	RB_CS_SysIO.qSTART	:=FALSE;
	eCSStatus:=E_CS_Status.EStop;	
END_IF
IF NOT RB_CS_SysIO.iEXT_CONTROL THEN
	eCSStatus:=E_CS_Status.LocalControl;	
END_IF
//
IF state<> 0 THEN
	eCSStatus:=E_CS_Status.Offline;
END_IF
// =====================================================
// BG
// =====================================================
tmrBGRun(IN:=  RB_CS_PickIO.cmd_wIndex <> RB_CS_PickIO.fb_wIndex,PT:= T#1s);
IF RB_CS_PickIO.cmd_wIndex = RB_CS_PickIO.fb_wIndex THEN
	RB_CS_PickIO.cmd_wIndex	:= RB_CS_PickIO.cmd_wIndex + 1;
	IF RB_CS_PickIO.cmd_wIndex > 255 THEN
		RB_CS_PickIO.cmd_wIndex:= 1;
	END_IF
END_IF


// =====================================================
// Mathod
// =====================================================

IF NOT _bLoadingDoneScan THEN
	_LoadingDoneScan	:= 0;
	tmrSimuLoadingDelay(IN:=FALSE);
END_IF


_bLoadingDoneScan:=FALSE;




IF NOT _bPickUpScan THEN
	_PickUpScan	:= 0;
	tmrSimuPickupDelay(IN:=FALSE);
END_IF



_bPickUpScan:=FALSE;

IF NOT _bPOUrun THEN
	_POUrun	:= 0;
	tmrPouRun(IN:=FALSE);
END_IF


_bPOUrun:=FALSE;






IF NOT _bInit THEN
	_Init:= 0;
END_IF


_bInit:= FALSE;

PROPERTY CommandError : BOOL
GET
CommandError	:= _Init = 99 OR _POUrun = 99;
END_GET
END_PROPERTY

METHOD Initialization : BOOL
VAR_INPUT
END_VAR
_bInit	:= TRUE;
CASE _Init OF
	0:
		tmrInit(IN:=FALSE);
		IF RB_CS_SysIO.iREADY THEN
			_Init	:= 5;
			ELSE
			RB_CS_SysIO.qENABLE	:= FALSE;
			_Init	:= 99;	
		END_IF
	5:
		RB_CS_SysIO.qENABLE	:= TRUE;
		tmrInit(IN:=FALSE,PT:= T#1S);
		IF RB_CS_SysIO.iENABLED THEN
			tmrInit(IN:=FALSE);
			_Init	:= 10;
		END_IF
		IF tmrInit.Q THEN
			tmrInit(IN:=FALSE);
			_Init	:= 99;
		END_IF
	
	10:
		IF RB_CS_SysIO.iRUNNING THEN
			_Init	:= 15;
			ELSE
			_Init	:= 30;	
		END_IF
	
	
		IF RB_CS_SysIO.iHome_Pos THEN
			tmrInit(IN:=FALSE);
			_Init	:= 50;
		END_IF;		
	15://取消程序
		RB_CS_SysIO.qRESET	:= TRUE;
		RB_CS_SysIO.qSTOP	:= TRUE;
		_Init				:= 16;
	16:
		tmrInit(IN:=FALSE,PT:= T#1S);
		IF NOT RB_CS_SysIO.iRUNNING THEN
			tmrInit(IN:=FALSE);
			RB_CS_SysIO.qRESET	:= FALSE;
			RB_CS_SysIO.qSTOP	:= FALSE;
			_Init				:= 30;
		END_IF
		IF tmrInit.Q THEN
			tmrInit(IN:=FALSE);
			_Init	:= 99;
		END_IF		

			
	30://RUN HOME
		RB_CS_SysIO.qPGNO	:= 61;
		RB_CS_SysIO.qSTART	:= TRUE;
		_Init				:= 31;
	31:
		tmrInit(IN:=NOT RB_CS_SysIO.iRUNNING,PT:= T#1S);		
		IF RB_CS_SysIO.iHome_Pos THEN
			RB_CS_SysIO.qSTART	:= FALSE;
			tmrInit(IN:=FALSE);
			_Init	:= 50;	
		END_IF
	
		IF RB_CS_SysIO.iPAUSED THEN
			RB_CS_SysIO.qCONTINUE:= TRUE;
		END_IF
	
		IF RB_CS_SysIO.iERROR OR tmrInit.q THEN
			tmrInit(IN:=FALSE);
			_Init	:= 99;
		END_IF
	99:
		;	
		
END_CASE;
(*
CASE _Init OF
0:
	RB_CS_SysIO.qENABLE	:= TRUE;
	tmrInit(IN:=FALSE);
	CASE eCSStatus OF
		E_CS_Status.Idle,E_CS_Status.EStop :
			_Init:= 99;
		E_CS_Status.DriveReady:
			_Init:= 50;
	    E_CS_Status.ReadyToWork:
			_Init:= 50;
	    E_CS_Status.Pou_Runing:
			_Init:= 11;
	    E_CS_Status.Pou_Run_Pause:
			_Init:= 11;
	    E_CS_Status.Pou_Run_Down:
			_Init:= 50;
	    E_CS_Status.Error:	
			_Init:= 10;		
	END_CASE
1:
	tmrInit(IN:=TRUE,PT:= T#0.5S);
	IF tmrInit.Q THEN
		wInitilRetry	:= wInitilRetry + 1;
		_Init:= 0;	
	END_IF
	
10://Error Reset
	RB_CS_SysIO.qRESET			:= TRUE;
	RB_CS_SysIO.qACKNOWLEDGEMSG	:= TRUE;
	_Init:= 1;
11://POU OFF
	RB_CS_SysIO.qSTOP			:= TRUE;
	_Init:= 1;	
50:
	tmrInit(IN:=FALSE);
	IF RB_CS_SysIO.iHome_Pos THEN
		_Init:= 90;
		ELSE
		_Init:= 55;
	END_IF
55:
	RB_CS_SysIO.qPGNO			:= 61;
	RB_CS_SysIO.qSTART			:= TRUE;
	RB_CS_PickIO.cmd_Velo		:= 20;
	_Init			:= 56;
56:
	CASE eCSStatus OF
		 E_CS_Status.Pou_Run_Down:
			_Init:= 50;		
		E_CS_Status.ReadyToWork	:
			_Init:= 50;
		 E_CS_Status.Error:	
		 	_Init:= 99;
	END_CASE;
		
90:
	Initialization	:= TRUE;
	
99:
;


   
    

END_CASE

*)
END_METHOD

ACTION IO_Mapp:
IF state <> 0 THEN
	;
END_IF

aryEIPOutput[0].0:=	RB_CS_SysIO.qSTOP		;	       
aryEIPOutput[0].1:=	RB_CS_SysIO.qSTART		;      
aryEIPOutput[0].2:=	RB_CS_SysIO.qPAUSE		;        
aryEIPOutput[0].3:=	RB_CS_SysIO.qCONTINUE	;      
aryEIPOutput[0].4:=	RB_CS_SysIO.qRESET		;        
aryEIPOutput[0].5:=  RB_CS_SysIO.qENABLE		;       
aryEIPOutput[0].6:=  RB_CS_SysIO.qPGNO.0		;
aryEIPOutput[0].7:=  RB_CS_SysIO.qPGNO.1			;       
aryEIPOutput[0].8:=  RB_CS_SysIO.qPGNO.2			;       
aryEIPOutput[0].9:=  RB_CS_SysIO.qPGNO.3			;       
aryEIPOutput[0].10:= RB_CS_SysIO.qPGNO.4			;       
aryEIPOutput[0].11:= RB_CS_SysIO.qPGNO.5			;	      
aryEIPOutput[0].12:= RB_CS_SysIO.qACKNOWLEDGEMSG	;
aryEIPOutput[0].13:= RB_CS_SysIO.qOVERRIDE		; 
aryEIPOutput[1].0	:=  RB_CS_PickIO.cmd_bBoxInPos;
aryEIPOutput[1].1	:=  RB_CS_PickIO.cmd_bPartInPos;
aryEIPOutput[1].8	:= RB_CS_PickIO.cmd_Velo.0;
aryEIPOutput[1].9	:= RB_CS_PickIO.cmd_Velo.1;
aryEIPOutput[1].10	:= RB_CS_PickIO.cmd_Velo.2;
aryEIPOutput[1].11	:= RB_CS_PickIO.cmd_Velo.3;
aryEIPOutput[1].12	:= RB_CS_PickIO.cmd_Velo.4;
aryEIPOutput[1].13	:= RB_CS_PickIO.cmd_Velo.5;
aryEIPOutput[1].14	:= RB_CS_PickIO.cmd_Velo.6;
aryEIPOutput[1].15	:= RB_CS_PickIO.cmd_Velo.7;

MEMCPY(ADR(aryEIPOutput[2]),ADR(RB_CS_PickIO.cmd_wIndex),1);



//

RB_CS_SysIO. iREADY    			:=   aryEIPInput[0].0;
RB_CS_SysIO. iRUNNING      		:=	 aryEIPInput[0].1;
RB_CS_SysIO. iPAUSED       		:=	 aryEIPInput[0].2;
RB_CS_SysIO. iSTOPPED      		:=	 aryEIPInput[0].3;
RB_CS_SysIO. iERROR        		:=	 aryEIPInput[0].4;
RB_CS_SysIO. iSAFEGURAD_ON 		:=	 aryEIPInput[0].5;
RB_CS_SysIO. iESTOP_ON     		:=	 aryEIPInput[0].6;
RB_CS_SysIO. iSERROR			:=	 aryEIPInput[0].7;
RB_CS_SysIO. iWARING            :=	 aryEIPInput[0].8;
RB_CS_SysIO. iENABLED         :=	 aryEIPInput[0].9;
RB_CS_SysIO. iACKNOWLEDGED    :=	 aryEIPInput[0].10;
RB_CS_SysIO. iERROR_CODE       :=	 aryEIPInput[0].11;
RB_CS_SysIO. iOVER_RIDE_OUT    :=	 aryEIPInput[0].12;
RB_CS_SysIO.iHome_Pos			:= aryEIPInput[3].0;
RB_CS_SysIO.iEXT_CONTROL			:= aryEIPInput[3].1;


RB_CS_PickIO.fb_bPacking		:= aryEIPInput[1].0;
RB_CS_PickIO.fb_bPackFinish		:= aryEIPInput[1].1;
RB_CS_PickIO.fb_putting			:= aryEIPInput[1].2;
RB_CS_PickIO.fb_PutFinish		:= aryEIPInput[1].3;
RB_CS_PickIO.fb_PackLayer.0		:= aryEIPInput[1].8;
RB_CS_PickIO.fb_PackLayer.1		:= aryEIPInput[1].9;
RB_CS_PickIO.fb_PackLayer.2		:= aryEIPInput[1].10;
RB_CS_PickIO.fb_PackLayer.3		:= aryEIPInput[1].11;

MEMCPY(ADR(RB_CS_PickIO.fb_Velo),ADR(aryEIPInput[2]),1);
MEMCPY(ADR(RB_CS_PickIO.fb_wIndex),ADR(aryEIPInput[2])+1,1);

//RB_CS_PickIO.cmd_Velo	:= RunParameter.Load_RBVelo;
END_ACTION

METHOD LoadingDone : BOOL
VAR_INPUT
END_VAR
_bLoadingDoneScan	:= TRUE;

IF Hmi_bBoxAutoTest THEN
	tmrSimuLoadingDelay(IN:= TRUE , PT:= Hmi_bBoxAutoTestTime);
	LoadingDone	:= tmrSimuLoadingDelay.q;
END_IF

IF NOT Hmi_bBoxAutoTest THEN
	CASE _LoadingDoneScan OF
		0:
			RB_CS_PickIO.cmd_bBoxInPos	:= TRUE;
			_LoadingDoneScan	:= 5;
		5:
			IF RB_CS_PickIO.fb_PutFinish THEN
				RB_CS_PickIO.cmd_bBoxInPos	:= FALSE;
				_LoadingDoneScan	:= 10;
			END_IF;		
		10:
			IF NOT RB_CS_PickIO.fb_PutFinish THEN
				_LoadingDoneScan	:= 15;
			END_IF;					
		15:
			LoadingDone:= TRUE;		
	END_CASE
END_IF;
END_METHOD

METHOD PickUp : BOOL
VAR_INPUT
END_VAR
_bPickUpScan:=TRUE;


IF Hmi_bPickAutoTest THEN
	tmrSimuPickupDelay(IN:= TRUE,PT:= Hmi_bPickAutoTestTime);
	PickUp	:=  tmrSimuPickupDelay.Q ;
END_IF;		
/////////
IF NOT Hmi_bPickAutoTest THEN
	CASE _PickUpScan OF
		0:
			RB_CS_PickIO.cmd_bPartInPos	:= TRUE;
			_PickUpScan	:= 5;
		5:
			IF RB_CS_PickIO.fb_bPackFinish	THEN
				RB_CS_PickIO.cmd_bPartInPos	:= FALSE;
				_PickUpScan	:= 10;
			END_IF
		10:
			IF NOT RB_CS_PickIO.fb_bPackFinish	THEN
				_PickUpScan	:= 15;
			END_IF				
		15:
			PickUp:= TRUE;		
	END_CASE
END_IF;

IF Hmi_bPickFeedTest THEN
	RB_CS_PickIO.cmd_bPartInPos	:= FALSE;
	Hmi_bPickFeedTest:=FALSE;
	PickUp	:= TRUE;
END_IF
END_METHOD

METHOD POU_Run : BOOL
VAR_INPUT
	Numb		:WORD;
END_VAR
VAR_OUTPUT
	Working		:BOOL;
	failRetrun	:BOOL;
END_VAR
_bPOUrun := TRUE;
CASE _POUrun OF
	0:
		RB_CS_SysIO.qRESET	:= FALSE;
		RB_CS_SysIO.qSTART	:= FALSE;
		RB_CS_PickIO.cmd_bBoxInPos	:=FALSE;
		RB_CS_PickIO.cmd_bPartInPos	:=FALSE;
		tmrPouRun(IN:=FALSE);
		wRetry				:= 0;
			CASE eCSStatus OF
				E_CS_Status.Idle :
					_POUrun:= 99;
				E_CS_Status.DriveReady:
					_POUrun:= 5;
			    E_CS_Status.ReadyToWork:
					_POUrun:= 10;
					IF Numb=0 THEN
						strTextBox:='Wait To Call';
						_POUrun:= 90;
					END_IF
			    E_CS_Status.Pou_Runing:
					_POUrun:= 90;
			    E_CS_Status.Pou_Run_Pause:
					_POUrun:= 90;
			    E_CS_Status.Pou_Run_Down:
					_POUrun:= 10;
					IF Numb=0 THEN
						strTextBox:='Wait To Call';
						_POUrun:= 90;
					END_IF
				E_CS_Status.EStop:
					_POUrun:= 99;
			    E_CS_Status.Error:	
					_POUrun:= 50;		
			END_CASE
	5:
			tmrPouRun(IN:= TRUE,PT:=T#1S);
			RB_CS_SysIO.qENABLE	:= TRUE;
			IF RB_CS_SysIO.iENABLED THEN
				_POUrun:= 0;
			END_IF
			IF tmrPouRun.Q THEN
				wRetry			:= wRetry+1;
				RB_CS_SysIO.qENABLE	:= FALSE;
				tmrPouRun(IN:=FALSE);
				_POUrun:= 6;
			END_IF
	6:
			tmrPouRun(IN:= TRUE,PT:=T#0.5S);
			IF tmrPouRun.Q THEN
				tmrPouRun(IN:=FALSE);
				_POUrun:= 5;
				IF wRetry >2 THEN
					strTextBox:='ENABLE Faild';
					_POUrun:= 98;	
				END_IF
			END_IF				
			
	10:
			tmrPouRun(IN:= TRUE,PT:=T#1S);
			RB_CS_SysIO.qPGNO:= WORD_TO_BYTE(Numb);
			RB_CS_SysIO.qSTART	:= TRUE;
			IF RB_CS_SysIO.iRUNNING THEN
				strTextBox:='Running';
				tmrPouRun(IN:= FALSE);
				_POUrun:= 90;
			END_IF
			IF Numb>65 THEN
				tmrPouRun(IN:= FALSE);
				strTextBox:='Numb. Out of Range';
				_POUrun:= 98;
			END_IF
			IF tmrPouRun.Q THEN
				strTextBox:='Star Time Out';
				_POUrun:= 98;
				tmrPouRun(IN:= FALSE);
			END_IF
	50://Error Reset
		tmrPouRun(IN:= TRUE,PT:=T#1S);	
		RB_CS_SysIO.qRESET	:= TRUE;
		IF eCSStatus<>  E_CS_Status.Error THEN
			strTextBox:='ERROR Reset';
			tmrPouRun(IN:= FALSE,PT:=T#1S);	
			_POUrun:= 10;
		END_IF
		
			IF tmrPouRun.Q THEN
				strTextBox:='Reset Faild';
				_POUrun:= 98;
				tmrPouRun(IN:= FALSE);
			END_IF	
	90://成功
		POU_Run	:= TRUE;
	
	98:
		
	99://失敗
		failRetrun:= TRUE;
		strTextBox:='Disallowed status';





END_CASE
END_METHOD

END_FUNCTION_BLOCK

// ---- 02_Unit/04_Kuka/RB_KR_Stacking.TcPOU
FUNCTION_BLOCK RB_KR_Stacking
VAR_INPUT
	state			AT%I*	:UINT;
	aryEIPInput		AT%I*	:ARRAY [0..127] OF BYTE ;
END_VAR

VAR_OUTPUT
	aryEIPOutput		AT%Q*	:ARRAY [0..127] OF BYTE ;
	strTextBox			:STRING(50);
	eKRStatus				:E_CS_Status;
	bOffline			:BOOL;
END_VAR
VAR
	_bCapture			:BOOL;
	_CaptureStep		:INT;
	_bPOUrun,_bPickUpScan,_bInit	:BOOL;
	_POUrun,_PickUpScan	,_InitStep			:INT;	
	tmrCapture			:TON;
	strText				:STRING;
	rPGNO_REQ			:R_TRIG;	
	tmrDriverReadyOnPulse,tmrConfMessOnPulse,tmrExtStarOnPulse	:TON;
	tmrPouRun,tmrForceExtStarOff: TON;
	tmrBGRun: TON;
	wRetry: INT;
END_VAR

IO_Mapp();
// =====================================================
// I/O
// =====================================================

tmrDriverReadyOnPulse(IN:=RB_KR_SysIO.qDRIVES_ON,PT:= T#0.3S);
IF tmrDriverReadyOnPulse.Q THEN
	RB_KR_SysIO.qDRIVES_ON	:=FALSE;
END_IF

tmrConfMessOnPulse(IN:= RB_KR_SysIO.qCONF_MESS,PT:=T#0.3S);
IF tmrConfMessOnPulse.Q THEN
	RB_KR_SysIO.qCONF_MESS:=FALSE;
END_IF

tmrExtStarOnPulse(IN:=RB_KR_SysIO.qEXT_START,PT:=T#0.3S);
IF tmrExtStarOnPulse.Q THEN
	RB_KR_SysIO.qEXT_START:=FALSE;
END_IF;
IF tmrForceExtStarOff.Q THEN
	tmrForceExtStarOff.IN:= FALSE;
END_IF



rPGNO_REQ(CLK:= RB_KR_SysIO.iPGNO_REQ);
IF rPGNO_REQ.Q THEN
	;
END_IF

// =====================================================
// FLAG
// =====================================================

IF NOT RB_KR_SysIO.iEXT_CONTROL THEN
	eKRStatus:= E_CS_Status.LocalControl;
	
	ELSE
	IF RB_KR_SysIO.iDRIVES_READY THEN
		eKRStatus:= E_CS_Status.DriveReady;
		
		IF	RB_KR_SysIO.iCONTROL_READY THEN
				eKRStatus:= E_CS_Status.DriverOn;
			IF RB_KR_SysIO.iPGNO_REQ THEN
				eKRStatus:= E_CS_Status.ReadyToWork;
			END_IF
			IF NOT RB_KR_SysIO.iRobotHomePos THEN
				eKRStatus:= E_CS_Status.LessHome;
			END_IF

		END_IF
		IF RB_KR_SysIO.iRobotRunning THEN
			eKRStatus:= E_CS_Status.Pou_Runing;
			IF RB_KR_SysIO.iPGNO_REQ THEN
				eKRStatus:= E_CS_Status.ReadyToWork;
			END_IF
		END_IF			
		
		IF RB_KR_SysIO.iSTOP_MESS THEN
			eKRStatus:= E_CS_Status.StopMess;
		END_IF		

			
		ELSE
		eKRStatus:= E_CS_Status.Idle;
	END_IF
END_IF

tmrBGRun(IN:=  RB_KR_StackingIO.cmd_wIndex <> RB_KR_StackingIO.fb_wIndex,PT:= T#1S);
IF RB_KR_StackingIO.cmd_wIndex = RB_KR_StackingIO.fb_wIndex THEN
	RB_KR_StackingIO.cmd_wIndex	:= RB_KR_StackingIO.cmd_wIndex + 1;
	IF RB_KR_StackingIO.cmd_wIndex > 255 THEN
		RB_KR_StackingIO.cmd_wIndex:= 1;
	END_IF
END_IF
























IF NOT _bCapture THEN
	_CaptureStep	:=0;

END_IF

_bCapture	:= FALSE;

//
IF NOT _bPOUrun THEN
	_POUrun	:=0;
END_IF

_bPOUrun:=FALSE;

METHOD Capture : BOOL
VAR_INPUT
END_VAR
_bCapture	:= TRUE;

CASE _CaptureStep OF
	0:
		RB_KR_StackingIO.cmd_bPartInPos	:= TRUE;
		_CaptureStep	:= 5;
		
	5:
		IF RB_KR_StackingIO.fb_bPickFinish THEN
			RB_KR_StackingIO.cmd_bPartInPos	:= FALSE;
			_CaptureStep	:= 10;
		END_IF

	10:
		IF NOT RB_KR_StackingIO.fb_bPickFinish THEN
			_CaptureStep	:= 15;
		END_IF		
	15:
		Capture:= TRUE;
END_CASE
END_METHOD

METHOD Initialization : BOOL
VAR_INPUT
END_VAR
_bInit	:= TRUE;

CASE _InitStep OF
	0:
		RB_KR_SysIO.qPGNO			:= 0;
		RB_KR_SysIO.qDRIVES_OFF		:= TRUE;
		RB_KR_SysIO.qMOVE_ENABLE	:= TRUE;
		RB_KR_SysIO.qCONF_MESS		:=  RB_KR_SysIO.iSTOP_MESS;
		_InitStep:= 5;
		
	5:
		CASE eKRStatus OF
				E_CS_Status.Idle :
					_InitStep:= 10;
				E_CS_Status.DriveReady:
					_InitStep:= 11;
				E_CS_Status.DriverOn:
					_InitStep:= 50;
			    E_CS_Status.ReadyToWork:
					_InitStep:= 50;
				E_CS_Status.StopMess:
					_InitStep:= 12;
			    E_CS_Status.Pou_Runing:
					_InitStep:= 90;
			    E_CS_Status.Pou_Run_Pause:
					_InitStep:= 90;
			    E_CS_Status.Pou_Run_Down:
					_InitStep:= 50;
	
			END_CASE
	10:
		RB_KR_SysIO.qDRIVES_ON:= TRUE;
		_InitStep:= 5;

	11:
	
		RB_KR_SysIO.qEXT_START:= TRUE;
		_InitStep:= 5;
		wRetry	:= wRetry + 1 ;
	12:
		RB_KR_SysIO.qEXT_START:= TRUE;
		RB_KR_SysIO.qCONF_MESS:= TRUE;
		_InitStep:= 5;
	50:
		Initialization:=TRUE;		
		

END_CASE
END_METHOD

ACTION IO_Mapp:
bOffline :=  state<>0 ;


aryEIPOutput[0].0:= RB_KR_SysIO.qDRIVES_ON	 ;  
aryEIPOutput[0].1:= RB_KR_SysIO.qDRIVES_OFF	  ;
aryEIPOutput[0].2:= RB_KR_SysIO.qMOVE_ENABLE;
aryEIPOutput[0].3:= RB_KR_SysIO.qCONF_MESS	 ;
aryEIPOutput[0].4:= RB_KR_SysIO.qEXT_START	 ;
//90為測試模式 
aryEIPOutput[0].5:= RB_KR_SysIO.qPgno.0;		     
aryEIPOutput[0].6:= RB_KR_SysIO.qPgno.1;	
aryEIPOutput[0].7:= RB_KR_SysIO.qPgno.2;
aryEIPOutput[1].0:= RB_KR_SysIO.qPgno.3;
aryEIPOutput[1].1:= RB_KR_SysIO.qPgno.4;
aryEIPOutput[1].2:= RB_KR_SysIO.qPgno.5;
aryEIPOutput[1].3:= RB_KR_SysIO.qPgno.6;
aryEIPOutput[1].4:= RB_KR_SysIO.qPgno.7;
					

aryEIPOutput[2].0:=	RB_KR_StackingIO.cmd_bPallet_AllowPut;				//棧板定位	
aryEIPOutput[2].1:= RB_KR_StackingIO.cmd_bReady;		       
aryEIPOutput[2].2:=	RB_KR_StackingIO.cmd_bCount0;			      
aryEIPOutput[2].3:=	RB_KR_StackingIO.cmd_bFence;	
		       
MEMCPY(ADR(aryEIPOutput[3]),ADR(RB_KR_StackingIO.cmd_wSize_length),2);
MEMCPY(ADR(aryEIPOutput[5]),ADR(RB_KR_StackingIO.cmd_wSize_width),2);
MEMCPY(ADR(aryEIPOutput[7]),ADR(RB_KR_StackingIO.cmd_wSize_height),2);
MEMCPY(ADR(aryEIPOutput[9]),ADR(RB_KR_StackingIO.cmd_wLayer_No),1);
   		     
aryEIPOutput[10].0	:=  RB_KR_StackingIO.cmd_bPartInPos	;	    		//取香訊號 
aryEIPOutput[10].1	:=  RB_KR_StackingIO.cmd_bSetting2Box	;   


MEMCPY(ADR(aryEIPOutput[11]),ADR(RB_KR_StackingIO.cmd_wIndex),1);
MEMCPY(ADR(aryEIPOutput[12]),ADR(RB_KR_StackingIO.cmd_Velo),1);

 
///////////////////////////////////////////////////////////////
RB_KR_SysIO.	iEXT_CONTROL		:= aryEIPInput[0].0;
RB_KR_SysIO.	iCONTROL_READY		:= aryEIPInput[0].1;
RB_KR_SysIO.	iSTOP_MESS			:= aryEIPInput[0].2;
RB_KR_SysIO.	iDRIVES_READY		:= aryEIPInput[0].3;
RB_KR_SysIO.	iPGNO_REQ			:= aryEIPInput[0].4;
RB_KR_SysIO.	iRobotHomePos		:= aryEIPInput[0].5;
RB_KR_SysIO.	iRobotRunning		:= aryEIPInput[0].6;
MEMCPY(ADR(RB_KR_StackingIO.fb_wPartNo),ADR(aryEIPInput[5]),1);
RB_KR_StackingIO.fb_bPickFinish				:= aryEIPInput[4].0;
RB_KR_StackingIO.fb_bWorking				:= aryEIPInput[4].1;
RB_KR_StackingIO.fb_bPalletFinish			:= aryEIPInput[4].2;
RB_KR_StackingIO.fb_bPalletInPos			:= aryEIPInput[4].3;
RB_KR_StackingIO.fb_wIndex					:=aryEIPInput[11] ;          
RB_KR_StackingIO.fb_bError[0]				:=aryEIPInput[6].0;	//曾數異常
MEMCPY(ADR(RB_KR_StackingIO.fb_wProNo),ADR(aryEIPInput[7]),1);





RB_KR_StackingIO.cmd_wSize_height	:= RunParameter.StackingRB_height;
RB_KR_StackingIO.cmd_wSize_length	:= RunParameter.StackingRB_length;
RB_KR_StackingIO.cmd_wSize_width	:= RunParameter.StackingRB_width;
RB_KR_StackingIO.cmd_bSetting2Box	:= RunParameter.stack_bUsed;
END_ACTION

METHOD POU_Run : BOOL
VAR_INPUT
	Numb		:WORD;
END_VAR
_bPOUrun	:= TRUE;

CASE _POUrun OF
	0:
		RB_KR_SysIO.qDRIVES_ON:= TRUE;
		RB_KR_SysIO.qMOVE_ENABLE:= TRUE;
		RB_KR_StackingIO.cmd_bCount0	:=FALSE;
		RB_KR_StackingIO.cmd_bPartInPos	:= FALSE;
		tmrPouRun(IN:= FALSE,PT:=T#1S);	

		CASE eKRStatus OF
				E_CS_Status.Idle :
					_POUrun:= 4;
				E_CS_Status.DriveReady:
					_POUrun:= 5;
				E_CS_Status.DriverOn:
					_POUrun:= 10;
					IF Numb=0 THEN
						strTextBox:='Wait To Call';
						_POUrun:= 90;
					END_IF
			    E_CS_Status.ReadyToWork:
					_POUrun:= 10;
					IF Numb=0 THEN
						strTextBox:='Wait To Call';
						_POUrun:= 90;
					END_IF
				E_CS_Status.StopMess:
						_POUrun:= 6;
			    E_CS_Status.Pou_Runing:
					_POUrun:= 90;
			    E_CS_Status.Pou_Run_Pause:
					_POUrun:= 90;
			    E_CS_Status.Pou_Run_Down:
					_POUrun:= 10;
					IF Numb=0 THEN
						strTextBox:='Wait To Call';
						_POUrun:= 90;
					END_IF
	
			END_CASE
	4:
		RB_KR_SysIO.qDRIVES_ON:= TRUE;
		_POUrun:= 7;

	5:
	
		RB_KR_SysIO.qEXT_START:= TRUE;
		_POUrun:= 7;
		wRetry	:= wRetry + 1 ;
	6:
		RB_KR_SysIO.qEXT_START:= TRUE;
		RB_KR_SysIO.qCONF_MESS:= TRUE;
		_POUrun:= 7;


	7:
		tmrPouRun(IN:= TRUE,PT:=T#0.5S);	
		IF tmrPouRun.Q THEN
			tmrPouRun(IN:= FALSE);
			_POUrun:= 0;
		END_IF			
	10:
			tmrPouRun(IN:= TRUE,PT:=T#1S);
			RB_KR_SysIO.qPGNO:= WORD_TO_BYTE(Numb);
			RB_KR_SysIO.qEXT_START	:= TRUE;
			IF RB_KR_SysIO.iRobotRunning THEN
				strTextBox:='Running';
				tmrPouRun(IN:= FALSE);
				_POUrun:= 90;
			END_IF
			IF Numb>95 THEN
				tmrPouRun(IN:= FALSE);
				strTextBox:='Numb. Out of Range';
				_POUrun:= 98;
			END_IF
			IF tmrPouRun.Q THEN
				strTextBox:='Star Time Out';
				_POUrun:= 98;
				tmrPouRun(IN:= FALSE);
			END_IF		
	
	90://完成
		POU_Run	:=TRUE;
	99://fail
		;
END_CASE
END_METHOD

END_FUNCTION_BLOCK

// ---- 02_Unit/99_Other/Spacil_FC.TcPOU
{attribute 'hide_all_locals'}
FUNCTION_BLOCK Spacil_FC
VAR_INPUT
END_VAR
VAR_OUTPUT
	SystemTime			:DT;
	ScanCounter			:DWORD;
	SM400	:BOOL;			// Alway TRUE
	SM401	:BOOL;			// Alway FALSE
	SM402	:BOOL;			// First Scan
	SM403	:BOOL;			// Secend Scan
	SM410	:BOOL;			// 0.1 Sec blinking
	SM411	:BOOL;			// 0.2 Sec blinking
	SM412	:BOOL;			// 1.0 Sec blinking
	SM413	:BOOL;			// 2.0 Sec blinking
	CpuUsage          	 :UDINT;
END_VAR
VAR
	_aryTmr			:ARRAY [0..10] OF TON;
	_IntenalHeart	:DWORD;
	fbLocalSystemTime:FB_LocalSystemTime := (bEnable := TRUE);
	timeAsDT        : DT;
	bRegi			:ARRAY [0..99] OF BOOL;
	wBuffer			:ARRAY [0..99] OF DWORD;
	i				:INT;
	fbCpuUsage:TC_CpuUsage;
END_VAR

ScanCounter	:= ScanCounter+1;
SM402	:= NOT SM400;
SM403	:= NOT SM402 ;
SM400	:= TRUE;
SM401	:= FALSE;
//SM410 0.1s
_aryTmr[0](IN:= TRUE , PT:= T#50MS);
IF _aryTmr[0].q  THEN
	_aryTmr[0](IN:= FALSE);
	SM410	:= NOT SM410;
END_IF
//SM411 0.2s
_aryTmr[1](IN:= TRUE , PT:= T#100MS);
IF _aryTmr[1].q  THEN
	_aryTmr[1](IN:= FALSE);
	SM411	:= NOT SM411;
END_IF
//SM412 1.0s
_aryTmr[2](IN:= TRUE , PT:= T#500MS);
IF _aryTmr[2].q  THEN
	_aryTmr[2](IN:= FALSE);
	SM412	:= NOT SM412;
END_IF
//sm413 2.0s
_aryTmr[3](IN:= TRUE , PT:= T#1S);
IF _aryTmr[3].q  THEN
	_aryTmr[3](IN:= FALSE);
	SM413	:= NOT SM413;
END_IF
fbLocalSystemTime();
SystemTime:= SYSTEMTIME_TO_DT(fbLocalSystemTime.systemTime);
fbCpuUsage(START:=SM410,USAGE=>CpuUsage);

METHOD GetOvertime : Time
VAR_INPUT
	mark	: INT;	//
END_VAR
VAR
	_CurrentCounter,_disCounter	:DWORD;
END_VAR
 _CurrentCounter :=ScanCounter;
 IF  wBuffer[mark] <> 0 THEN
	 
	IF _CurrentCounter >  wBuffer[mark] THEN
		_disCounter	:=  _CurrentCounter -  wBuffer[mark];
		ELSE
		_disCounter	:=   wBuffer[mark] - _CurrentCounter;	
	END_IF
	
	
	 GetOvertime:= DWORD_TO_TIME(_disCounter);
END_IF;

 wBuffer[mark]	:= _CurrentCounter;
END_METHOD

METHOD GetOvertime_Clear : BOOL
VAR_INPUT
	mark	: INT;	//
END_VAR
 wBuffer[mark]	:= 0;
END_METHOD

METHOD GetOvertime_Renew : Time
VAR_INPUT
	mark	: INT;	//
END_VAR
VAR
	_CurrentCounter,_disCounter	:DWORD;
END_VAR
 _CurrentCounter :=ScanCounter;
 wBuffer[mark]	:= _CurrentCounter;
END_METHOD

END_FUNCTION_BLOCK

// ---- 02_Unit/01_Customization/MainControl.TcPOU
FUNCTION_BLOCK MainControl
VAR_INPUT
END_VAR
VAR_OUTPUT
END_VAR
VAR
	MC_Stop:ARRAY [1..6] OF MC_Stop;	
	_bStop			:BOOL;
	i	 			:INT;
	fbMC_UngroupAllAxes	: MC_UngroupAllAxes;
	fbMC_GroupDisable	: MC_GroupDisable;
	fbAddAxis			: ARRAY[1..2] OF MC_AddAxisToGroup;
	fbMC_GroupEnable	: MC_GroupEnable;	
	_bDual_Release		:BOOL;
	nReleaseStep		:INT;
	_bReset				:BOOL;

END_VAR

MC_Stop[1](Axis:= Axis_FlyIn);
MC_Stop[2](Axis:= Axis_DualServo1);
MC_Stop[3](Axis:= Axis_DualServo2);
MC_Stop[4](Axis:= Axis_BoxPullOut);
MC_Stop[5](Axis:= Axis_load1);
MC_Stop[6](Axis:= Axis_load2);

FOR i := 1TO 6 DO
	IF MC_Stop[i].Done OR MC_Stop[i].Error THEN
		MC_Stop[i].Execute	:= FALSE;
	END_IF
END_FOR;



_bStop :=FALSE;


IF Setting_FanAuto THEN
	Fan();
END_IF


//

fbAddAxis[1](AxesGroup:=DualGroupRef, Axis := Axis_DualServo1);
fbAddAxis[2](AxesGroup:=DualGroupRef, Axis := Axis_DualServo2);
fbMC_GroupDisable(AxesGroup:=DualGroupRef);
IF fbMC_GroupDisable.Done OR fbMC_GroupDisable.Error THEN
	fbMC_GroupDisable.Execute:= FALSE;
END_IF



_bDual_Release	:=FALSE;
//RESET






_bReset:= FALSE;

METHOD Dual_Release : BOOL
VAR_INPUT
END_VAR
_bDual_Release	:= TRUE;

CASE nReleaseStep OF
	0:
		IF Axis_DualServo1.Status.DiscreteMotion THEN
			fbAddAxis[1].Execute:=TRUE;
			fbAddAxis[2].Execute:=TRUE;
		END_IF



	



END_CASE
END_METHOD

METHOD ErrorReset : BOOL
VAR_INPUT
END_VAR
Cyl_AxisBoxCatch.bReset	:= TRUE;
Cyl_BoxSideBottom.bReset	:= TRUE;
Cyl_Axis90.bReset		:= TRUE;
Cyl_AxisBottom.bReset	:= TRUE;
Cyl_UnloadDef.bReset	:= TRUE;

IF Axis_DualServo1.Status.Error THEN
	Axis_DualServo1.Reset();
END_IF
IF Axis_DualServo2.Status.Error THEN
	Axis_DualServo2.Reset();
END_IF
IF Axis_BoxPullOut.Status.Error THEN
	Axis_BoxPullOut.Reset();
END_IF
IF Axis_load1.Status.Error THEN
	Axis_load1.Reset();
END_IF
IF Axis_load2.Status.Error THEN
	Axis_load2.Reset();
END_IF
IF Axis_FlyIn.Status.Error THEN
	Axis_FlyIn.Reset();
END_IF
END_METHOD

METHOD Fan : BOOL
VAR_INPUT
END_VAR
TemperatureFans:=TemperatureHigh;
END_METHOD

METHOD ResetAllAxes : BOOL
VAR_INPUT
END_VAR
Axis_DualServo1.Reset();
Axis_DualServo2.Reset();
Axis_FlyIn.Reset();
END_METHOD

METHOD SoftStopAxis : BOOL
VAR_INPUT
END_VAR
IF Axis_BoxPullOut.Status.Moving THEN
	Axis_BoxPullOut.Stop();
END_IF
IF Axis_DualServo1.Status.Moving THEN
	Axis_DualServo1.Stop();
END_IF
IF Axis_DualServo2.Status.Moving THEN
	Axis_DualServo2.Stop();
END_IF
IF Axis_FlyIn.Status.Moving THEN
	Axis_FlyIn.Stop();
END_IF
IF Axis_load1.Status.Moving THEN
	Axis_load1.Stop();
END_IF
IF Axis_load2.Status.Moving THEN
	Axis_load2.Stop();
END_IF
IF DualGroupRef.NcToPlc.CA.common.GroupStatus.State = mcGroupStateMoving THEN
	fbMC_GroupDisable(AxesGroup:= DualGroupRef,Execute:= TRUE);
END_IF
END_METHOD

METHOD StopAir : BOOL
VAR_INPUT
END_VAR

Cyl_BoxSidePitch	.qExtendCoil	:= FALSE;
Cyl_BoxSideBottom	.qExtendCoil	:= FALSE;
Cyl_AxisBoxCatch	.qExtendCoil	:= FALSE;
Vacm_AxisCatchBox					:= FALSE;					
Cyl_Axis90			.qExtendCoil	:= FALSE;		
Vacm_Axis90							:= FALSE;	
Cyl_AxisBottom		.qExtendCoil	:= FALSE;	
Cyl_BeltBottom		.qExtendCoil	:= FALSE;	
Cyl_BeltBottomSup	.qExtendCoil	:= FALSE;	
Cyl_UnloadDef		.qExtendCoil	:= FALSE;	
Cyl_NGPurge			.qExtendCoil	:= FALSE;	
Cyl_ShockStop		.qExtendCoil	:= FALSE;	
Cyl_StackUD			.qExtendCoil	:= FALSE;	
Cyl_ExitClip		.qExtendCoil	:= FALSE;	
Cyl_ExitStopper		.qExtendCoil	:= FALSE;	
Cyl_FlyIn_Pass						:= FALSE;
END_METHOD

METHOD StopAllAxes : BOOL
VAR_INPUT
END_VAR
_bStop	:= TRUE;

FOR i := 1TO 6 DO
	MC_Stop[i].Execute	:= TRUE;
END_FOR;
END_METHOD

METHOD StopMotor : BOOL
VAR_INPUT
END_VAR
Motor_LoadIn.qRun			:=FALSE;						
Motor_Blower.qRun			:=FALSE;							
Motor_LoadPurge1.qRun		:=FALSE;	
Motor_LoadPurge2.qRun		:=FALSE;	
Motor_BoxSealBottom_L.qRun	:=FALSE;
Motor_BoxSealBottom_R.qRun	:=FALSE;
Roller_Purge.qRun			:=FALSE;							
Roller_Exit.qRun			:=FALSE;		
Motor_shock.qRun			:=FALSE;
END_METHOD

END_FUNCTION_BLOCK

// ---- 01_POUs/static/MST_POU.TcPOU
PROGRAM MST_POU	//Mechanical structure testing
VAR
	bDualRingCycleTest	:BOOL;
	dualtestVelo		:REAL;
	nStep				:INT;
	strText				:STRING(50);

	//
	tmrDelay			:TON;
	MC_GearIn			:MC_GearIn;
	MC_Stop				: MC_Stop;
	MC_MoveVelocity		: MC_MoveVelocity := (Velocity := 100);
	fbTrigger_Load1	,	fbTrigger_Load2			:R_TRIG;
	Loadin1Pos		:ARRAY [1..10] OF LREAL ;
	Loadin2Pos		:ARRAY [1..10] OF LREAL ;
	i					:INT;
	
	//
	M	:ARRAY [0..50] OF BOOL ;
	D	:ARRAY [0..50] OF INT := [60, 90, 49(0)] ;
	MC_TouchProbeDual1,MC_TouchProbeDual2,MC_TouchProbeFly: MC_TouchProbe;
	TouchTriggerDual1,TouchTriggerDual2,TouchTriggerFly	:TRIGGER_REF;
	MC_AbortTrigger1,MC_AbortTrigger2					: MC_AbortTrigger;
	fbLDF		:ARRAY [0..50] OF F_TRIG;
	//Loadcell Check
	bLoadcell_MaxLoad , bLoadcell_RefLoad ,bLoadcell_Percent ,bLoadcell_fbcmd ,bLoadTara ,bLoadcell_ZeroCali ,bLoadcell_Loadcail	:BOOL;
	tmrLoadcellfbcmd	:TON;
END_VAR

IF PB_EMG OR OP.xInitialRuning OR OP.xAutoRuning THEN
	FOR i:= 0 TO 50 DO
		M[i]:=FALSE;
	END_FOR
END_IF



IF M[0] THEN
	M[6]:= M_DualServo.Initialization(M[1]);
	IF M[6] THEN
		M[0]	:=FALSE;
	END_IF
END_IF
fbLDF[0](CLK:= M[0]);
IF fbLDF[0].Q THEN
	IF Axis_DualServo1.Status.Moving THEN
		Axis_DualServo1.Reset();
	END_IF
	IF Axis_DualServo2.Status.Moving THEN
		Axis_DualServo2.Reset();
	END_IF
END_IF


IF M[4] THEN
	MainControl.SoftStopAxis();
END_IF
IF M[5] THEN
	M_DualServo.Process(FALSE);
END_IF

fbLDF[5](CLK:= M[5]);
IF fbLDF[5].Q THEN
	Motor_LoadIn.qRun:=FALSE;
	Cyl_FlyIn_Pass:=FALSE;
END_IF;


fbTrigger_Load1(CLK:= Sen_AxisLoad1ORG);
fbTrigger_Load2(CLK:= Sen_AxisLoad2ORG);
IF fbTrigger_Load1.Q THEN
	FOR i := 9 TO 1 BY -1 DO
		Loadin1Pos[i+1]:= Loadin1Pos[i];
	END_FOR
	Loadin1Pos[1]	:= Axis_load1.NcToPlc.ActPos;
END_IF

IF fbTrigger_Load2.Q THEN
	FOR i := 9 TO 1 BY -1 DO
		Loadin2Pos[i+1]:= Loadin2Pos[i];
	END_FOR
	Loadin2Pos[1]	:= Axis_load2.NcToPlc.ActPos;
END_IF

//開箱 
IF M[10] THEN
	M[12]:=FALSE;
	M[11]:=M_Openbox1.Initialization(FALSE);
END_IF;
IF M[11] THEN
	M[10]:=FALSE;
END_IF;
IF M[12] THEN
	M[10]:=FALSE;
	M[11]:=M_Openbox1.Process(M[13]);
END_IF;
IF M[14] THEN
	M_Openbox1.HaltStepContiune();
	M[14]:=FALSE;
END_IF;
		
//裝箱  
IF M[15] THEN
	M[16]:=M_LoadPic3.Initialization(FALSE);
END_IF;
IF M[16] THEN
	M[15]:=FALSE;
END_IF;
IF M[16] THEN
	M[15]:=FALSE;
END_IF;
IF M[17] THEN
	M[16]:=M_LoadPic3.Process(M[18]);
END_IF;
IF M[19] THEN
	M_LoadPic3.HaltStepContiune();
	M[19]:=FALSE;
END_IF;

//封箱底  
IF M[20] THEN
	M[22]	:=FALSE;
	M[21]:=M_Sealing2.Initialization(FALSE);
END_IF;
IF M[21] THEN
	M[20]:=FALSE;
END_IF;
IF M[22] THEN
	M[20]	:=FALSE;
	M[21]:=M_Sealing2.Process(M[23]);
END_IF;
IF M[24] THEN
	M_Sealing2.HaltStepContiune();
	M[24]:=FALSE;
END_IF;

//秤重晃   
IF M[25] THEN
	M[26]:=M_UnloadNG4.Initialization(FALSE);
END_IF;
IF M[26] THEN
	M[25]:=FALSE;
END_IF;
IF M[27] THEN
	M[26]:=M_UnloadNG4.Process(M[28]);
END_IF;
IF M[29] THEN
	M_UnloadNG4.HaltStepContiune();
	M[29]:=FALSE;
END_IF;

//堆疊

IF M[30] THEN
	M[31]:=M_StackComv5.Initialization(FALSE);
END_IF;
IF M[31] THEN
	M[30]:=FALSE;
END_IF;
IF M[32] THEN
	M[31]:=M_StackComv5.Process(FALSE);
END_IF;
//堆疊手臂

IF M[35] THEN
	M[36]:=M_RBStack6.Initialization(FALSE);
END_IF;
IF M[37] THEN
	M[36]:=M_RBStack6.Process(M[38]);
END_IF;
IF M[39] THEN
	M_RBStack6.HaltStepContiune();
	M[39]:=FALSE;
END_IF;

IF M[40] THEN
	MainControl.StopAllAxes();
	M[40]:=FALSE;
END_IF

IF M[41] THEN
	 M[42]:=RB_CS.Initialization();
END_IF

IF M[43] THEN
	 M[42]:=RB_CS.POU_Run(INT_TO_BYTE(D[0]));
END_IF

IF M[44] THEN
	 M[45]:=RB_KR.POU_Run(INT_TO_BYTE(D[1]));
END_IF
IF M[46] THEN
	 M[45]	:=	RB_KR.Initialization();
END_IF



//Loadcell
IF bLoadcell_MaxLoad THEN
	bLoadcell_fbcmd	:=LoadCell.SetNomialLoad(Setting_MaxLoad);
END_IF

IF bLoadcell_RefLoad THEN
	bLoadcell_fbcmd	:=LoadCell.SetRefLoad(Setting_RefLoad);

END_IF

IF bLoadcell_Percent THEN
	bLoadcell_fbcmd	:=LoadCell.SetScaleFactor(Setting_LoadPercent);
END_IF

IF bLoadcell_ZeroCali THEN
	bLoadcell_fbcmd	:=LoadCell.SetZeroCalibration();
END_IF

IF bLoadcell_Loadcail THEN
	bLoadcell_fbcmd	:=LoadCell.SetLoadCalibration();
END_IF

